// TIA Portal V17 export
// export: Created 2024-09-02T12:50:16.2754473Z, ExportSetting WithDefaults, DisplayName Totally Integrated Automation Portal, DisplayVersion V17, DisplayName TIA Portal Openness, DisplayVersion V17, DisplayName TIA Portal Version Control Interface, DisplayVersion V17, DisplayName STEP 7 Professional, DisplayVersion V17, DisplayName STEP 7 Safety, DisplayVersion V17, DisplayName WinCC Professional, DisplayVersion V17
DATA_BLOCK "AnwDB_ZP_Alarm_OP70"   // DB255
{ S7_Optimized_Access := 'TRUE'; DB_Accessible_From_OPC_UA := 'FALSE' }
AUTHOR : OlegFuehrus
FAMILY : BA
NAME : BA
VERSION : 0.1
// stored: AutoNumber false, DBAccessibleFromOPCUA false, IsOnlyStoredInLoadMemory false, IsRetainMemResEnabled false, IsWriteProtectedInAS false, MemoryReserve 100
   VAR
      FAULT : Array[1..1024] of Bool;
      WARNING : Array[1..1024] of Bool;
      INFORMATION : Array[1..256] of Bool;
      FaultsNo_ST1 : Int;
      FaultsNoSK_ST1 : Int;
      ReportsNo_ST1 : Int;
      FaultsNo_ST2 : Int;
      FaultsNoSK_ST2 : Int;
      ReportsNo_ST2 : Int;
      FaultsNo_ST3 : Int;
      FaultsNoSK_ST3 : Int;
      ReportsNo_ST3 : Int;
   END_VAR
BEGIN
   // FAULT[1] : ESB: Steuerspannung fehlt [+S01- BG0.1]] / Alarm 1: Controle Voltage Not OK [+S01- BG0.1]] / Alarm 1: Stuurspanning niet in(+S01-600KF0.1 of +S01-111KF3) [+S01- BG0.1]]
   // FAULT[2] : ESB: Profibus-Teilnehmer gestört
   // FAULT[3] : ESB: ProfiNet-Teilnehmer gestört / Alarm 3: ProfiNet - Member fault / Alarm 3: ProfiNet - Deelnemerfout
   // FAULT[4] : ESB: Einschaltbedingung fehlt / Alarm 4: switch-on condition missing / Alarm 4: Inschakelvoorwaarde ontbreekt
   // FAULT[5] : ESB: Pneumatikdruck n.i.O. [+M01- BG50.7] / Alarm 5: Pneumatic pressure on OP70 NIO [+M01- BG50.7] / Alarm 5: Pneumatische druk OP70 NIO [+M01- BG50.7]
   // FAULT[6] : ESB: Sicherungsfall 24V [ -100TB1-100FC3/6/8 , [+S01- BG0.2]] / Alarm 6: 24V fuse fault [ -100TB1-100FC3/6/8 , [+S01- BG0.2]] / Alarm 6: 24V-zekeringfout [ -100TB1-100FC3/6/8 , [+S01- BG0.2]]
   // FAULT[7] : ESB: Sicherungsfall 230V [-33FC1/-33FB4/6 -44FC1/3, [+S01- BG0.3]] / Alarm 7: 230V fuse fault [-33FC1/-33FB4/6 -44FC3,-45FC1/3/5, [+S01- BG0.3]] / Alarm 7: 230V-zekeringfout [-33FC1/-33FB4/6 -44FC3,-45FC1/3/5, [+S01- BG0.3]]
   // FAULT[8] : ESB: Sicherungsfall 400V [-30QB7-50QB3,[+S01- BG0.4]] / Alarm 8: 400V fuse fault [-30QB7, [+S01- BG0.4]] / Alarm 8: 400V-zekeringfout[-30QB7, [+S01- BG0.4]]
   // FAULT[9] : ESB: Sicherungsfall 230V ....... [+S-QBxxx]
   // FAULT[10] : ESB: Sicherungsfall 230V ....... [+S-QBxxx]
   // FAULT[11] : ESB: kein Text
   // FAULT[12] : ESB: kein Text
   // FAULT[13] : ESB: kein Text
   // FAULT[14] : ESB: kein Text
   // FAULT[15] : ESB: kein Text
   // FAULT[16] : ESB: kein Text
   // FAULT[17] : ESB: kein Text
   // FAULT[18] : ESB: kein Text
   // FAULT[19] : ESB: kein Text
   // FAULT[20] : ESB: kein Text
   // FAULT[21] : ESB: kein Text
   // FAULT[22] : ESB: kein Text
   // FAULT[23] : ESB: kein Text
   // FAULT[24] : ESB: kein Text
   // FAULT[25] : Allg: Nacharbeit in Station aktiv / Alarm 25: Reworking in Station / Alarm 25: Rework in Station
   // FAULT[26] : Allg: Moby 1 Störung VorStopper [+M01-17BX1] / Alarm 26: RFID 1 fault prestopper [+M01-17BX1] / Alarm 26: Voorstopper RFID 1 fout [+M01-17BX1]
   // FAULT[27] : Allg: Moby 2 Störung Stopper [+M01-17BX2] / Alarm 27: RFID 2 fault Stopper [+M01-17BX2] / Alarm 27: Stopper RFID 2 fout [+M01-17BX2]
   // FAULT[28] : Allg: Moby 3 Störung Stopper [+M01-17BX2] / Alarm 28: RFID 3 fault Stopper [+M01-17BX2] / Alarm 28: Stopper RFID 3 fout [+M01-17BX2]
   // FAULT[29] : Allg: Moby 4 Störung Stopper XXXXX [+M01-BX606]
   // FAULT[30] : Allg: Moby 5 Störung Stopper XXXXX [+M01-BX608]
   // FAULT[31] : Allg: Moby 6 Störung Stopper XXXXX [+M01-BX610]
   // FAULT[32] : Allg: kein Text
   // FAULT[33] : Allg: Pneumatikdruck n.i.O. Station [+M01 - BG700.0/1] / Alarm 33: Central Pneumatic fault [+M01- BG50.7] / Alarm 33: Pneumatische toevoer storing OP70 [+M01- BG50.7]
   // FAULT[34] : Allg: Pneumatikdruck n.i.O. Roboter 1 [+M01 - BG707.0/1] / Alarm 34: Pneumatic ON Gripper fault [+M01- BG53.7] / Alarm 34: Pneumatische toevoer storing OP70 - grijper [+M01- BG53.7]
   // FAULT[35] : Allg: Pneumatikdruck n.i.O. Roboter 2 [+M01 - BG707.2/3]
   // FAULT[36] : Allg: Pneumatikdruck n.i.O. Reserve
   // FAULT[37] : Allg: kein Text
   // FAULT[38] : Allg: kein Text
   // FAULT[39] : Allg: kein Text
   // FAULT[40] : Allg: kein Text
   // FAULT[41] : Allg: kein Text
   // FAULT[42] : Allg: Temperatur Schaltschrank (>30 Minuten) überschritten [+S01--300BT0.7] / Alarm 42: Control cabinet temperature exceeded (> 30 minutes) [+S01--300BT0.7] / Alarm 42: Temperatuur schakelkast overschreden (> 30 minuten) [+S01--300BT0.7]
   // FAULT[43] : Allg: kein Text
   // FAULT[44] : Allg: kein Text
   // FAULT[45] : Allg: Alarm Netzgerät vor Maschine Ein [+S01-600KF0.1] / Alarm 45: Power supply in Machine On Alarm [+S01-600KF0.1] / Alarm 45: Stuurspanning niet in [+S01-600KF0.1]
   // FAULT[46] : Allg: Störung ProfiNet Switch -275XF1 [+S01- BG0.5] / Alarm 46: Fault in ProfiNet Switch -275XF1 [+S01- BG0.5] / Alarm 46: Storing in ProfiNet Switch -275XF1 [+S01- BG0.5]
   // FAULT[47] : Allg: kein Text
   // FAULT[48] : Allg: Grundstellungsfahrt erforderlich / Alarm 48: Home required not allowed / Alarm 48: HOME positie rijden niet toegestaan
   // FAULT[49] : Safety: NOT-HALT Hauptbedienpult OP 40 gestört [+ZP01-302SF30.0] / Alarm 49: EMERGENCY STOP Main Panel OP70[+ZP01-302SF30.0] / Alarm 49: NOODSTOP HMI OP 70[+ZP01-302SF30.0]
   // FAULT[50] : Safety: NOT-HALT Hauptbedienpult OP 50 gestört [+ZP01-11SF5] / Alarm 50: EMERGENCY STOP Main Panel OP 50[+ZP01-11SF5] / Alarm 50: NOODSTOP HMI OP 70[+ZP01-11SF5]
   // FAULT[51] : Safety: NOT-HALT Schutztür XXXXXX gestört [+M01-SF320]
   // FAULT[52] : Safety: NOT-HALT Schutztür XXXXXX gestört [+M01-SF 340]
   // FAULT[53] : Safety: NOT-HALT Roboter 1 gestört [+R01-SF 1]
   // FAULT[54] : Safety: NOT-HALT Roboter 2 gestört [+R02-SF 1]
   // FAULT[55] : Safety: NOT-HALT Reserve
   // FAULT[56] : Safety: NOT-HALT Reserve
   // FAULT[57] : Safety: NOT-HALT Reserve
   // FAULT[58] : Safety: NOT-HALT Reserve
   // FAULT[59] : Safety: NOT-HALT Reserve
   // FAULT[60] : Safety: NOT-HALT Reserve
   // FAULT[61] : Safety: NOT-HALT Reserve
   // FAULT[62] : Safety: NOT-HALT Reserve
   // FAULT[63] : Safety: NOT-HALT Reserve
   // FAULT[64] : Safety: NOT-HALT nicht quittiert OP40 / Alarm 64: EMERGENCY STOP MAIN PANEL OP70 not acknowledged / Alarm 64: NOODSTOP HMI OP 70 niet bevestigd
   // FAULT[65] : Safety: NOT-HALT nicht quittiert OP50 / Alarm 65: EMERGENCY STOP MAIN PANEL OP50 not acknowledged / Alarm 65: NOODSTOP HMI OP70 niet bevestigd
   // FAULT[66] : Safety: Schutztür Station offen [+M01-30SF0] / Alarm 66: Safety Door opened [+M01-260SF2] / Alarm 66: Veiligheidsdeur geopend OP70 [+M01-260SF0]
   // FAULT[67] : Safety: Schutztür Station offen [+M01-SF210.1]
   // FAULT[68] : Safety: Schutztür Station offen [+M01-SFxxxx]
   // FAULT[69] : Safety: Schutztür Reserve
   // FAULT[70] : Safety: Schutztür Reserve
   // FAULT[71] : Safety: Schutztür Reserve
   // FAULT[72] : Safety: Schutztür Reserve
   // FAULT[73] : Safety: Schutztür Reserve
   // FAULT[74] : Safety: Schutztür Reserve
   // FAULT[75] : Safety: Schutztür Reserve
   // FAULT[76] : Safety: Schutztür Reserve
   // FAULT[77] : Safety: Schutztür Reserve
   // FAULT[78] : Safety: Schutztür Reserve
   // FAULT[79] : Safety: Schutztür Reserve
   // FAULT[80] : Safety: Schutztür Reserve
   // FAULT[81] : Safety: Schutztür Station nicht quittiert
   // FAULT[82] : Safety: Schutztür Station nicht quittiert
   // FAULT[83] : Safety: Schutztür Station nicht quittiert / Alarm 83: Safety Door not acknowledged / Alarm 83: Veiligheidsdeur gesloten OP70 niet bevestigd
   // FAULT[84] : Safety: Lichtgitter WT Einlauf ausgelöst (Muting)
   // FAULT[85] : Safety: Lichtgitter WT Auslauf ausgelöst (Muting)
   // FAULT[86] : Safety: Lichtgitter Reserve
   // FAULT[87] : Safety: Lichtgitter Reserve
   // FAULT[88] : Safety: Lichtgitter Reserve
   // FAULT[89] : Safety: Lichtgitter Reserve
   // FAULT[90] : Alarm 90: Safety Bolts Sensor not active, Bolts insite / Alarm 90: Sensor veiligheidsbouten niet actief, bouten op locatie
   // FAULT[91] : Safety: Lichtgitter Reserve
   // FAULT[92] : Safety: Lichtgitter Reserve
   // FAULT[93] : Safety: Lichtgitter Reserve
   // FAULT[94] : Safety: Lichtgitter Reserve
   // FAULT[95] : Safety: Lichtgitter Reserve
   // FAULT[96] : Safety: Lichtgitter Reserve
   // FAULT[97] : Safety: Lichtgitter WT Einlauf nicht quittiert (Muting)
   // FAULT[98] : Safety: Lichtgitter WT Auslauf nicht quittiert (Muting)
   // FAULT[99] : Safety: Freigabekreise gestört
   // FAULT[100] : Safety: Freigabekreis 1 gestört - Medien einschalten
   // FAULT[101] : Safety: Freigabekreis 1 gestört - Sicherheit Station NIO / Alarm 101: Safety Feedback Circuit 1 - Enabling safety Circuit OP70 NOK / Alarm 101: Veiligheidsfeedbackcircuit 1 - inschakelen van veiligheidscircuit OP70 NOK
   // FAULT[102] : Safety: Freigabekreis 2 gestört - Not Halt NIO / Alarm 102: Safety Feedback Circuit 2 - Enabling safety Circuit 2(Emergency stop) NOK / Alarm 102: Veiligheidsfeedbackcircuit 2 - inschakelen van veiligheidscircuit 2 (noodstop) NOK
   // FAULT[103] : Safety: Freigabekreis 4 gestört -
   // FAULT[104] : Safety: Freigabekreis 5 gestört -
   // FAULT[105] : Safety: Freigabekreis 6 gestört -
   // FAULT[106] : Safety: Freigabekreis 7 gestört -
   // FAULT[107] : Safety: Freigabekreis 8 gestört -
   // FAULT[108] : Safety: Freigabekreis 9 gestört -
   // FAULT[109] : Safety: Freigabekreis 10 gestört -
   // FAULT[110] : Safety: Freigabekreis 11 gestört -
   // FAULT[111] : Safety: Freigabekreis 12 gestört -
   // FAULT[112] : Safety: Freigabekreis 13 gestört -
   // FAULT[113] : Safety: Freigabekreis 14 gestört
   // FAULT[114] : Safety: Freigabekreis 15 gestört
   // FAULT[115] : Safety: F-Baugruppenfehler: "F00030_-265KF5".QBAD / Alarm 115: Module error: "F00030_-265KF5".QBAD / Alarm 115: Profisafeodulefout: "F00030_-265KF5".QBAD
   // FAULT[116] : Safety: F-Baugruppenfehler: "F00036_-265KF6".QBAD / Alarm 116: Module error: "F00036_-265KF6".QBAD / Alarm 116: Profisafe modulefout: "F00036_-265KF6".QBAD
   // FAULT[117] : Safety: F-Baugruppenfehler: Reserve
   // FAULT[118] : Safety: F-Baugruppenfehler: Reserve
   // FAULT[119] : Safety: F-Baugruppenfehler: Reserve
   // FAULT[120] : Safety: F-Baugruppenfehler: Reserve
   // FAULT[121] : Safety: F-Baugruppenfehler: Reserve
   // FAULT[122] : Safety: F-Baugruppenfehler: Reserve
   // FAULT[123] : Safety: F-Baugruppenfehler: Reserve
   // FAULT[124] : Safety: F-Baugruppenfehler: Reserve
   // FAULT[125] : Safety: F-Baugruppenfehler: Reserve
   // FAULT[126] : Safety: F-Baugruppenfehler: Reserve
   // FAULT[127] : Safety: F-Baugruppenfehler: Reserve
   // FAULT[128] : Safety: F-Baugruppenfehler: Reserve
   // FAULT[129] : Safety: F-Baugruppenfehler: Reserve
   // FAULT[130] : Safety: F-Baugruppenfehler: Reserve
   // FAULT[131] : Safety: F-Baugruppenfehler: Reserve
   // FAULT[132] : Safety: F-Baugruppenfehler: Reserve
   // FAULT[133] : Safety: F-Baugruppenfehler: Reserve
   // FAULT[134] : Safety: F-Baugruppenfehler: Reserve
   // FAULT[135] : Safety: F-Baugruppenfehler: Reserve
   // FAULT[136] : Safety: F-Baugruppenfehler: Reserve
   // FAULT[137] : Safety: F-Baugruppenfehler: Reserve
   // FAULT[138] : Safety: F-Baugruppenfehler: Reserve
   // FAULT[139] : Safety: F-Baugruppenfehler: Reserve
   // FAULT[140] : Safety: F-Baugruppenfehler: Reserve
   // FAULT[141] : Safety: F-Baugruppenfehler: Reserve
   // FAULT[142] : Safety: F-Baugruppenfehler: Reserve
   // FAULT[143] : Safety: F-Baugruppenfehler: Reserve
   // FAULT[144] : Safety: kein Text
   // FAULT[145] : Safety: kein Text
   // FAULT[146] : Safety: kein Text
   // FAULT[147] : Safety: kein Text
   // FAULT[148] : Safety: kein Text
   // FAULT[149] : Safety: kein Text
   // FAULT[150] : Safety: kein Text
   // FAULT[151] : Safety: kein Text
   // FAULT[152] : Safety: kein Text
   // FAULT[153] : Safety: kein Text
   // FAULT[154] : Safety: kein Text
   // FAULT[155] : Safety: kein Text
   // FAULT[156] : Safety: kein Text
   // FAULT[157] : Safety: kein Text
   // FAULT[158] : Safety: kein Text
   // FAULT[159] : Safety: kein Text
   // FAULT[160] : Safety: Schutztür Reserve
   // FAULT[161] : Safety: kein Text
   // FAULT[162] : Safety: kein Text
   // FAULT[163] : Safety: kein Text
   // FAULT[164] : Safety: kein Text
   // FAULT[165] : Safety: kein Text
   // FAULT[166] : Safety: kein Text
   // FAULT[167] : Safety: kein Text
   // FAULT[168] : Safety: kein Text
   // FAULT[169] : Safety: kein Text
   // FAULT[170] : Safety: kein Text
   // FAULT[171] : Safety: kein Text
   // FAULT[172] : Safety: kein Text
   // FAULT[173] : Safety: kein Text
   // FAULT[174] : Safety: kein Text
   // FAULT[175] : Safety: kein Text
   // FAULT[176] : Safety: kein Text
   // FAULT[177] : Safety: Rückführkreisüberwachung Sicherheit Station NIO [E3.4] / Alarm 177: Feedback circuit monitoring Enabling safety Circuit 1 OP70 [+S01- BG3.4] / Alarm 177: Bewaking terugkoppelingscircuit veiligheid station OK OP70[+S01- BG3.4]
   // FAULT[178] : Safety: Rückführkreisüberwachung Not Halt NIO [E3.5] / Alarm 178: Feedback circuit monitoring EMERGENCY STOP Station [E3.5] / Alarm 178: Bewaking terugkoppelingscircuit noodstop OK OP70 [E3.5]
   // FAULT[179] : Safety: Rückführkreisüberwachung Luft NIO [E50.7] / Alarm 179: Feedback circuit monitoring Pneumatic NOK [+M01- BG50.7] / Alarm 179: Bewaking terugkoppelcircuit Pneumatisch NOK[+M01- BG50.7]
   // FAULT[180] : Safety: Rückführkreisüberwachung Luft im Greifer NIO [E53.7] / Alarm 180: Feedback circuit monitoring Pneumatic NOK in Gripper [+M01- BG53.7] / Alarm 180: Bewaking terugkoppelcircuit Pneumatisch NOK in grijper[+M01- BG53.7]
   // FAULT[181] : Safety: Rückführkreisüberwachung Reserve
   // FAULT[182] : Safety: Rückführkreisüberwachung Reserve
   // FAULT[183] : Safety: Rückführkreisüberwachung Reserve
   // FAULT[184] : Safety: Rückführkreisüberwachung mPro400SG fehlerhaft [E3.2]
   // FAULT[185] : Safety: Rückführkreisüberwachung Reserve
   // FAULT[186] : Safety: Rückführkreisüberwachung Vertikalachse Bremsen [QL712.0/1]
   // FAULT[187] : Safety: Rückführkreisüberwachung Reserve
   // FAULT[188] : Safety: Rückführkreisüberwachung Reserve
   // FAULT[189] : Safety: Rückführkreisüberwachung Reserve
   // FAULT[190] : Alarm 190: Feeder Unit Empty Damper Cap [I55.4] / Alarm 190: Demperdop van de invoereenheid leeg [I55.4]
   // FAULT[191] : Alarm 191: Feeder Unit Empty Ball [I56.0] / Alarm 191: Lege bal invoereenheid [I56.0]
   // FAULT[192] : Alarm 192: Feeder Unit Empty Screw [I56.1] / Alarm 192: Schroef invoereenheid leeg [I56.1]
   // FAULT[193] : Safety: Rückführkreisüberwachung Reserve
   // FAULT[194] : Safety: Rückführkreisüberwachung Reserve
   // FAULT[195] : Safety: Rückführkreisüberwachung Reserve
   // FAULT[196] : Safety: Rückführkreisüberwachung Reserve
   // FAULT[197] : Safety: Rückführkreisüberwachung Reserve
   // FAULT[198] : Safety: Rückführkreisüberwachung Reserve
   // FAULT[199] : Safety: Rückführkreisüberwachung Reserve
   // FAULT[200] : Safety: Rückführkreisüberwachung Reserve
   // FAULT[201] : Safety: Rückführkreisüberwachung Reserve
   // FAULT[202] : Safety: Rückführkreisüberwachung Reserve
   // FAULT[203] : Safety: Rückführkreisüberwachung Reserve
   // FAULT[204] : Safety: Rückführkreisüberwachung Reserve
   // FAULT[205] : Safety: Rückführkreisüberwachung Reserve
   // FAULT[206] : Safety: Rückführkreisüberwachung Reserve
   // FAULT[207] : Safety: Rückführkreisüberwachung Reserve
   // FAULT[208] : Safety: Rückführkreisüberwachung Reserve
   // FAULT[209] : Fehler Schmierzyklus - Automatik gesperrt
   // FAULT[210] : Allg: kein Text
   // FAULT[211] : Allg: kein Text
   // FAULT[212] : Allg: kein Text
   // FAULT[213] : Allg: kein Text
   // FAULT[214] : Allg: kein Text
   // FAULT[215] : Allg: kein Text
   // FAULT[216] : Allg: kein Text
   // FAULT[217] : Allg: kein Text
   // FAULT[218] : Allg: kein Text
   // FAULT[219] : Allg: kein Text
   // FAULT[220] : Allg: kein Text
   // FAULT[221] : Allg: kein Text
   // FAULT[222] : Allg: kein Text
   // FAULT[223] : Allg: kein Text
   // FAULT[224] : Allg: kein Text
   // FAULT[225] : Allg: kein Text
   // FAULT[226] : Allg: kein Text
   // FAULT[227] : Allg: kein Text
   // FAULT[228] : Allg: kein Text
   // FAULT[229] : Allg: kein Text
   // FAULT[230] : Allg: kein Text
   // FAULT[231] : Allg: kein Text
   // FAULT[232] : Allg: kein Text
   // FAULT[233] : Allg: kein Text
   // FAULT[234] : Allg: kein Text
   // FAULT[235] : Allg: kein Text
   // FAULT[236] : Allg: kein Text
   // FAULT[237] : Allg: kein Text
   // FAULT[238] : Allg: kein Text
   // FAULT[239] : Allg: kein Text
   // FAULT[240] : Allg: kein Text
   // FAULT[241] : Allg: kein Text
   // FAULT[242] : Allg: kein Text
   // FAULT[243] : Allg: kein Text
   // FAULT[244] : Allg: kein Text
   // FAULT[245] : Allg: kein Text
   // FAULT[246] : Allg: kein Text
   // FAULT[247] : Allg: kein Text
   // FAULT[248] : Allg: kein Text
   // FAULT[249] : Allg: kein Text
   // FAULT[250] : Allg: kein Text
   // FAULT[251] : Allg: kein Text
   // FAULT[252] : Allg: kein Text
   // FAULT[253] : Allg: kein Text
   // FAULT[254] : Allg: kein Text
   // FAULT[255] : Allg: kein Text
   // FAULT[256] : Allg: kein Text
   // FAULT[257] : Allg: kein Text
   // FAULT[258] : Allg: kein Text
   // FAULT[259] : Allg: kein Text
   // FAULT[260] : Allg: kein Text
   // FAULT[261] : Allg: kein Text
   // FAULT[262] : Allg: kein Text
   // FAULT[263] : Allg: kein Text
   // FAULT[264] : Allg: kein Text
   // FAULT[265] : Überwachung Schütz "Sinamics" nicht abgefallen bzw. defeckt (+S01-QA101.1)
   // FAULT[266] : Überwachung Schütz "Kühlgerät" nicht abgefallen bzw. defeckt (+S01-QA100.2)
   // FAULT[267] : Überwachung Schütz "Schmierung" nicht abgefallen bzw. defeckt (+S01-QA101.0)
   // FAULT[268] : Überwachung Schütz "Schraubtechnik" nicht abgefallen bzw. defeckt (+S01-QA102.0)
   // FAULT[269] : Überwachung Schütz " " nicht abgefallen Reserve
   // FAULT[270] : Überwachung Schütz " " nicht abgefallen Reserve
   // FAULT[271] : Überwachung Schütz " " nicht abgefallen Reserve
   // FAULT[272] : Überwachung Schütz " " nicht abgefallen Reserve
   // FAULT[273] : Überwachung Schütz " " nicht abgefallen Reserve
   // FAULT[274] : Überwachung Schütz " " nicht abgefallen Reserve
   // FAULT[275] : Allg: kein Text
   // FAULT[276] : Allg: kein Text
   // FAULT[277] : Allg: kein Text
   // FAULT[278] : Allg: kein Text
   // FAULT[279] : Allg: kein Text
   // FAULT[280] : Allg: kein Text
   // FAULT[281] : Allg: kein Text
   // FAULT[282] : Allg: kein Text
   // FAULT[283] : Allg: kein Text
   // FAULT[284] : Allg: kein Text
   // FAULT[285] : Allg: kein Text
   // FAULT[286] : Allg: kein Text
   // FAULT[287] : Allg: kein Text
   // FAULT[288] : Allg: kein Text
   // FAULT[289] : Allg: kein Text
   // FAULT[290] : Allg: kein Text
   // FAULT[291] : Allg: kein Text
   // FAULT[292] : Allg: kein Text
   // FAULT[293] : Allg: kein Text
   // FAULT[294] : Allg: kein Text
   // FAULT[295] : Allg: kein Text
   // FAULT[296] : Allg: kein Text
   // FAULT[297] : Serienfehler: BEA1 Lagerrahmen verschrauben - Schraubstelle 01 / SeriesError: FG01 BEA1 Assembly Damper Cap / Seriefout: FG01 BEA1 Montage demper cap
   // FAULT[298] : Serienfehler: BEA1 Lagerrahmen verschrauben - Schraubstelle 02 / SeriesError: FG01 BEA1 Assembly Ball / Seriefout: FG01 BEA1 Montage bal
   // FAULT[299] : Serienfehler: BEA1 Lagerrahmen verschrauben - Schraubstelle 03 / SeriesError: FG01 BEA2 Damper Cap controle / Seriefout: FG01 BEA2 Controle positie demper cap
   // FAULT[300] : Serienfehler: BEA1 Lagerrahmen verschrauben - Schraubstelle 04 / SeriesError: FG02 BEA1 Controle Damper 1 - OP50 / Seriefout: FG02 BEA1 Controle Demper 1 - OP50
   // FAULT[301] : Serienfehler: BEA1 Lagerrahmen verschrauben - Schraubstelle 05 / SeriesError: FG02 BEA1 Controle Damper 2 - OP50 / Seriefout: FG02 BEA1 Controle Demper 2 - OP50
   // FAULT[302] : Serienfehler: BEA1 Lagerrahmen verschrauben - Schraubstelle 06 / SeriesError: FG02 BEA1 Controle Damper 3 - OP50 / Seriefout: FG02 BEA1 Controle Demper 3 - OP50
   // FAULT[303] : Serienfehler: BEA1 Lagerrahmen verschrauben - Schraubstelle 07 / SeriesError: FG02 BEA1 Controle Filter - OP60 / Seriefout: FG02 BEA1 Controle filter - OP60
   // FAULT[304] : Serienfehler: BEA1 Lagerrahmen verschrauben - Schraubstelle 08 / SeriesError: FG02 BEA1 Controle Ball - OP70_1 / Seriefout: FG02 BEA1 Controle kogel - OP70_1
   // FAULT[305] : Serienfehler: BEA1 Lagerrahmen verschrauben - Schraubstelle 09 / SeriesError: FG02 BEA1 Controle Damper Cap - OP70_1 / Seriefout: FG02 BEA1 Controle Demper cap - OP70_1
   // FAULT[306] : Serienfehler: BEA1 Lagerrahmen verschrauben - Schraubstelle 10 / SeriesError: FG02 BEA1 ControleDowel 1 - OP60 / Seriefout: FG02 BEA2 Tussenplaat nemen
   // FAULT[307] : Serienfehler: BEA1 Lagerrahmen verschrauben - Schraubstelle 11 / SeriesError: FG02 BEA1 Controle Dowel 2 - OP60 / Seriefout: FG02 BEA2 Tussenplaat plaatsen
   // FAULT[308] : Serienfehler: BEA1 Lagerrahmen verschrauben - Schraubstelle 12 / SeriesError: FG02 BEA2 Pick Intermediate plate / Seriefout: FG02 BEA3 Tussenplaat vastdraaien
   // FAULT[309] : Serienfehler: BEA1 Lagerrahmen verschrauben - Schraubstelle 13 / SeriesError: FG02 BEA2 Place Intermediate plate
   // FAULT[310] : Serienfehler: BEA1 Lagerrahmen verschrauben - Schraubstelle 14 / SeriesError: FG02 BEA3 Tightening Intermediate plate
   // FAULT[311] : Serienfehler: BEA1 Lagerrahmen verschrauben - Schraubstelle 15
   // FAULT[312] : Serienfehler: BEA1 Lagerrahmen verschrauben - Schraubstelle 16
   // FAULT[313] : Serienfehler: BEA1 Lagerrahmen verschrauben - Schraubstelle 01
   // FAULT[314] : Serienfehler: BEA1 Lagerrahmen verschrauben - Schraubstelle 01
   // FAULT[315] : Serienfehler: Reserve
   // FAULT[316] : Serienfehler: Reserve
   // FAULT[317] : Serienfehler: Reserve
   // FAULT[318] : Serienfehler: Reserve
   // FAULT[319] : Serienfehler: Reserve
   // FAULT[320] : Serienfehler: Reserve
   // FAULT[321] : Serienfehler: Reserve
   // FAULT[322] : Serienfehler: Reserve
   // FAULT[323] : Serienfehler: Reserve
   // FAULT[324] : Serienfehler: Reserve
   // FAULT[325] : Serienfehler: Reserve
   // FAULT[326] : Serienfehler: Reserve
   // FAULT[327] : Serienfehler: Reserve
   // FAULT[328] : Serienfehler: Reserve
   // FAULT[329] : Allg: kein Text
   // FAULT[330] : Allg: kein Text
   // FAULT[331] : Allg: kein Text
   // FAULT[332] : Allg: kein Text
   // FAULT[333] : Allg: kein Text
   // FAULT[334] : Allg: kein Text
   // FAULT[335] : Allg: kein Text
   // FAULT[336] : Allg: kein Text
   // FAULT[337] : Allg: kein Text
   // FAULT[338] : Allg: kein Text
   // FAULT[339] : Allg: kein Text
   // FAULT[340] : Allg: kein Text
   // FAULT[341] : Paarfehler: MM30/31 Hub-index unten/oben(+M01-BG51.1/51.0) / Pair error: MM30/31 Index Up / Down(+M01-BG51.1/51.0) / Paarfout: MM30/31 Index Boven/Onder (+M01-BG51.1/51.0)
   // FAULT[342] : Paarfehler: MM50/51 Hub-index unten/oben(+M01-BG51.3-5/51.2-4) / Pair error: MM50/51 Index Up / Down(+M01-BG51.3-5/51.2-4) / Paarfout: MM50/51 Index Boven/Onder (+M01-BG51.3-5/51.2-4)
   // FAULT[343] : Paarfehler: MM70/71 Hub-index unten/oben(+M01-BG52.0/52.1) / Pair error: MM70/71 Index Up / Down(+M01-BG52.0/52.1) / Paarfout: MM70/71 Index Boven/Onder (+M01-BG52.0/52.1)
   // FAULT[344] : Pair error: MM110 Sliding Damper Cap Back/ Front (+M01-BG52.5/4) / Paarfehler: MM110 Schieber Kappe züruck/vor (+M01-BG52.5/4) / Paarfout: MM110 schuifdemperkap Vooraan/Achteraan (+M01-BG52.5/4)
   // FAULT[345] : Paarfehler: MM120 Schieber Kugel züruck/vor (+M01-BG53.0/1) / Pair error: MM120 Sliding Ball Back/ Front (+M01-BG53.0/1) / Paarfout: MM120 Sliding Ball Vooraan/Achteraan (+M01-BG53.0/1)
   // FAULT[346] : Paarfehler: MM130 Fügeeinheit Kappe senken/heben(+M01-BG53.3/4) / Pair error: MM130 Press Damper Cap Up/Down (+M01-BG53.3/4) / Paarfout: MM130 Druk demperkap Boven/Onder (+M01-BG53.3/4)
   // FAULT[347] : Paarfehler: MM140 Y-Achse Übersetzer züruck/vor(+M01-BG53.5/6) / Pair error: MM140 Y-Axis Gripper Back/ Front (+M01-BG53.5/6) / Paarfout: MM140 Y-as grijper Vooraan/Achteraan(+M01-BG53.5/6)
   // FAULT[348] : Paarfehler: MM160 Z-Achse Übersetzerl heben/senken (+M01-BG54.0/1) / Pair error: MM150 Z-Axis Gripper Up/Down (+M01-BG54.0/1) / Paarfout: MM150 Z-as grijper Boven/Onder (+M01-BG54.0/1)
   // FAULT[349] : Paarfehler: MM170 Hubzylinder Schraubeinheit heben/senken(+M01-BG54.2/3) / Pair error: MM160 Z-Axis Screwdriver Up/Down (+M01-BG54.2/3) / Paarfout: MM160 Z-as schroevendraaier Boven/Onder (+M01-BG54.2/3)
   // FAULT[350] : Paarfehler: MM180 Zustellschlitten heben/senken (+M01-BG54.4/5) / Pair error: MM170 Z-Axis Screwdriver unit Up/Down (+M01-BG54.4/5) / Paarfout: MM170 Z-as Schroevendraaiereenheid Boven/Onder (+M01-BG54.4/5)
   // FAULT[351] : Paarfehler: MM200 Übersetzen Hülse züruck/vor (+M01-BG63.0/1) / Pair error: MM210 Loading cylinder Dumper Cap Up/Down (+M01-BG55.0/1) / Paarfout: MM210 Laadcilinder Dumper Cap Boven/Onder (+M01-BG55.0/1)
   // FAULT[352] : Paarfehler: MM210 Zustellung Hülse züruck/vor (+M01-BG63.2/3) / Pair error: MM220 Separation cylinder Dumper Cap unit front/back (+M01-BG55.6/7) / Paarfout: MM220 Scheidingscilinder Dumper Cap unit Vooraan/Achteraan (+M01-BG55.6/7)
   // FAULT[353] : Paarfehler: *** reserviert für Paarfehler ***
   // FAULT[354] : Paarfehler: *** reserviert für Paarfehler ***
   // FAULT[355] : Paarfehler: *** reserviert für Paarfehler ***
   // FAULT[356] : Paarfehler: *** reserviert für Paarfehler ***
   // FAULT[357] : Paarfehler: *** reserviert für Paarfehler ***
   // FAULT[358] : Paarfehler: *** reserviert für Paarfehler ***
   // FAULT[359] : Paarfehler: *** reserviert für Paarfehler ***
   // FAULT[360] : Paarfehler: *** reserviert für Paarfehler ***
   // FAULT[361] : Paarfehler: *** reserviert für Paarfehler ***
   // FAULT[362] : Paarfehler: *** reserviert für Paarfehler ***
   // FAULT[363] : Paarfehler: *** reserviert für Paarfehler ***
   // FAULT[364] : Paarfehler: *** reserviert für Paarfehler ***
   // FAULT[365] : Paarfehler: *** reserviert für Paarfehler ***
   // FAULT[366] : Paarfehler: *** reserviert für Paarfehler ***
   // FAULT[367] : Paarfehler: *** reserviert für Paarfehler ***
   // FAULT[368] : Paarfehler: *** reserviert für Paarfehler ***
   // FAULT[369] : Paarfehler: *** reserviert für Paarfehler ***
   // FAULT[370] : Paarfehler: *** reserviert für Paarfehler ***
   // FAULT[371] : Paarfehler: *** reserviert für Paarfehler ***
   // FAULT[372] : Paarfehler: *** reserviert für Paarfehler ***
   // FAULT[373] : Paarfehler: *** reserviert für Paarfehler ***
   // FAULT[374] : Paarfehler: *** reserviert für Paarfehler ***
   // FAULT[375] : Paarfehler: *** reserviert für Paarfehler ***
   // FAULT[376] : Paarfehler: *** reserviert für Paarfehler ***
   // FAULT[377] : Paarfehler: *** reserviert für Paarfehler ***
   // FAULT[378] : Paarfehler: *** reserviert für Paarfehler ***
   // FAULT[379] : Paarfehler: *** reserviert für Paarfehler ***
   // FAULT[380] : Paarfehler: *** reserviert für Paarfehler ***
   // FAULT[381] : Paarfehler: *** reserviert für Paarfehler ***
   // FAULT[382] : Paarfehler: *** reserviert für Paarfehler ***
   // FAULT[383] : Paarfehler: *** reserviert für Paarfehler ***
   // FAULT[384] : Paarfehler: *** reserviert für Paarfehler ***
   // FAULT[385] : Paarfehler: *** reserviert für Paarfehler ***
   // FAULT[386] : Paarfehler: *** reserviert für Paarfehler ***
   // FAULT[387] : Paarfehler: *** reserviert für Paarfehler ***
   // FAULT[388] : Paarfehler: *** reserviert für Paarfehler ***
   // FAULT[389] : Paarfehler: *** reserviert für Paarfehler ***
   // FAULT[390] : Paarfehler: *** reserviert für Paarfehler ***
   // FAULT[391] : Paarfehler: *** reserviert für Paarfehler ***
   // FAULT[392] : Paarfehler: *** reserviert für Paarfehler ***
   // FAULT[393] : Paarfehler: *** reserviert für Paarfehler ***
   // FAULT[394] : Paarfehler: *** reserviert für Paarfehler ***
   // FAULT[395] : Paarfehler: *** reserviert für Paarfehler ***
   // FAULT[396] : Paarfehler: *** reserviert für Paarfehler ***
   // FAULT[397] : Paarfehler: *** reserviert für Paarfehler ***
   // FAULT[398] : Paarfehler: *** reserviert für Paarfehler ***
   // FAULT[399] : Paarfehler: *** reserviert für Paarfehler ***
   // FAULT[400] : Paarfehler: *** reserviert für Paarfehler ***
   // FAULT[401] : Paarfehler: *** reserviert für Paarfehler ***
   // FAULT[402] : Paarfehler: *** reserviert für Paarfehler ***
   // FAULT[403] : Paarfehler: *** reserviert für Paarfehler ***
   // FAULT[404] : Paarfehler: *** reserviert für Paarfehler ***
   // FAULT[405] : Paarfehler: *** reserviert für Paarfehler ***
   // FAULT[406] : Paarfehler: *** reserviert für Paarfehler ***
   // FAULT[407] : Paarfehler: *** reserviert für Paarfehler ***
   // FAULT[408] : Paarfehler: *** reserviert für Paarfehler ***
   // FAULT[409] : Paarfehler: *** reserviert für Paarfehler ***
   // FAULT[410] : Paarfehler: *** reserviert für Paarfehler ***
   // FAULT[411] : Paarfehler: *** reserviert für Paarfehler ***
   // FAULT[412] : Paarfehler: *** reserviert für Paarfehler ***
   // FAULT[413] : Paarfehler: *** reserviert für Paarfehler ***
   // FAULT[414] : Paarfehler: *** reserviert für Paarfehler ***
   // FAULT[415] : Paarfehler: *** reserviert für Paarfehler ***
   // FAULT[416] : Paarfehler: *** reserviert für Paarfehler ***
   // FAULT[417] : Fehler - Automatik gesperrt
   // FAULT[418] : Fehler - Automatik gesperrt
   // FAULT[419] : Fehler - Automatik gesperrt
   // FAULT[420] : Fehler - Automatik gesperrt
   // FAULT[421] : Fehler - Automatik gesperrt
   // FAULT[422] : Fehler - Automatik gesperrt
   // FAULT[423] : Fehler - Automatik gesperrt
   // FAULT[424] : Fehler - Automatik gesperrt
   // FAULT[425] : Achse: Vertikalschlitten - Motorschutz [+S01-QA1.1]
   // FAULT[426] : Achse: Vertikalschlitten - Störung [+S01-KF110]
   // FAULT[427] : Achse: Vertikalschlitten - Bremsentest n.i.O.
   // FAULT[428] : Achse: kein Text
   // FAULT[429] : Achse: kein Text
   // FAULT[430] : Achse: kein Text
   // FAULT[431] : Achse: kein Text
   // FAULT[432] : Achse: kein Text
   // FAULT[433] : Achse: kein Text
   // FAULT[434] : Achse: kein Text
   // FAULT[435] : Achse: kein Text
   // FAULT[436] : Achse: kein Text
   // FAULT[437] : Achse: kein Text
   // FAULT[438] : Achse: kein Text
   // FAULT[439] : Achse: kein Text
   // FAULT[440] : Achse: kein Text
   // FAULT[441] : Achse: kein Text
   // FAULT[442] : Achse: kein Text
   // FAULT[443] : Achse: kein Text
   // FAULT[444] : Achse: kein Text
   // FAULT[445] : Achse: kein Text
   // FAULT[446] : Achse: kein Text
   // FAULT[447] : Achse: kein Text
   // FAULT[448] : Achse: kein Text
   // FAULT[449] : Achse: kein Text
   // FAULT[450] : Achse: kein Text
   // FAULT[451] : Achse: kein Text
   // FAULT[452] : Achse: kein Text
   // FAULT[453] : Achse: kein Text
   // FAULT[454] : Achse: kein Text
   // FAULT[455] : Achse: kein Text
   // FAULT[456] : Achse: kein Text
   // FAULT[457] : Schrauber: MPRO 1 nicht Betriebsbereit [+M-KF100]
   // FAULT[458] : Schrauber: MPRO 1 Sicherungen ausgelöst [E1.4]
   // FAULT[459] : Schrauber: kein Text
   // FAULT[460] : Schrauber: kein Text
   // FAULT[461] : Schrauber: kein Text
   // FAULT[462] : Schrauber: kein Text
   // FAULT[463] : Schrauber: kein Text
   // FAULT[464] : Schrauber: kein Text
   // FAULT[465] : Schrauber: kein Text
   // FAULT[466] : Schrauber: kein Text
   // FAULT[467] : Schrauber: kein Text
   // FAULT[468] : Schrauber: kein Text
   // FAULT[469] : Schrauber: kein Text
   // FAULT[470] : Schrauber: kein Text
   // FAULT[471] : Schrauber: kein Text
   // FAULT[472] : Schrauber: kein Text
   // FAULT[473] : Allg: kein Text
   // FAULT[474] : Allg: kein Text
   // FAULT[475] : Allg: kein Text
   // FAULT[476] : Allg: kein Text
   // FAULT[477] : Allg: kein Text
   // FAULT[478] : Allg: kein Text
   // FAULT[479] : Allg: kein Text
   // FAULT[480] : Allg: kein Text
   // FAULT[481] : Allg: kein Text
   // FAULT[482] : Allg: kein Text
   // FAULT[483] : Allg: kein Text
   // FAULT[484] : Allg: kein Text
   // FAULT[485] : Allg: kein Text
   // FAULT[486] : Allg: kein Text
   // FAULT[487] : Allg: kein Text
   // FAULT[488] : Allg: kein Text
   // FAULT[489] : Allg: kein Text
   // FAULT[490] : Allg: kein Text
   // FAULT[491] : Allg: kein Text
   // FAULT[492] : Allg: kein Text
   // FAULT[493] : Allg: kein Text
   // FAULT[494] : Allg: kein Text
   // FAULT[495] : Allg: kein Text
   // FAULT[496] : Allg: kein Text
   // FAULT[497] : Allg: kein Text
   // FAULT[498] : Allg: kein Text
   // FAULT[499] : Allg: kein Text
   // FAULT[500] : Allg: kein Text / Alarm 500: X2 - The assumed level of NOK has been reached / Alarm 500: X2 - Het ingestelde niveau aantal NOK delen is bereikt
   // FAULT[501] : Allg: kein Text
   // FAULT[502] : Allg: kein Text
   // FAULT[503] : Allg: kein Text
   // FAULT[504] : Allg: kein Text
   // FAULT[505] : Allg: kein Text
   // FAULT[506] : Allg: kein Text
   // FAULT[507] : Allg: kein Text
   // FAULT[508] : Allg: kein Text
   // FAULT[509] : Allg: kein Text
   // FAULT[510] : Allg: kein Text
   // FAULT[511] : Allg: kein Text
   // FAULT[512] : Allg: kein Text
   // FAULT[513] : Roboter 1 - Greiferbewegung verklemmt [+R01]
   // FAULT[514] : Roboter 1 - Kollisionsschutz ausgelöst [+R01]
   // FAULT[515] : Roboter 1 - Fehler Teilekontrolle Greifer 1
   // FAULT[516] : Roboter 1 - Fehler Teilekontrolle Greifer 2
   // FAULT[517] : Roboter 1 -
   // FAULT[518] : Roboter 1 -
   // FAULT[519] : Roboter 1 -
   // FAULT[520] : Roboter 1 -
   // FAULT[521] : Roboter 1 -
   // FAULT[522] : Roboter 1 -
   // FAULT[523] : Roboter 1 -
   // FAULT[524] : Roboter 1 -
   // FAULT[525] : Roboter 1 -
   // FAULT[526] : Roboter 1 -
   // FAULT[527] : Roboter 1 -
   // FAULT[528] : Roboter 1 -
   // FAULT[529] : Roboter 2 - Greiferbewegung verklemmt [+R02]
   // FAULT[530] : Roboter 2 - Kollisionsschutz ausgelöst [+R02]
   // FAULT[531] : Roboter 2 - Fehler Teilekontrolle Greifer 1
   // FAULT[532] : Roboter 2 - Fehler Teilekontrolle Greifer 2
   // FAULT[533] : Roboter 2 -
   // FAULT[534] : Roboter 2 -
   // FAULT[535] : Roboter 2 -
   // FAULT[536] : Roboter 2 -
   // FAULT[537] : Roboter 2 -
   // FAULT[538] : Roboter 2 -
   // FAULT[539] : Roboter 2 -
   // FAULT[540] : Roboter 2 -
   // FAULT[541] : Roboter 2 -
   // FAULT[542] : Roboter 2 -
   // FAULT[543] : Roboter 2 -
   // FAULT[544] : Roboter 2 -
   // FAULT[545] : fehler545
   // FAULT[546] : fehler546
   // FAULT[547] : fehler547
   // FAULT[548] : fehler548
   // FAULT[549] : fehler549
   // FAULT[550] : fehler550
   // FAULT[551] : fehler551
   // FAULT[552] : fehler552
   // FAULT[553] : fehler553
   // FAULT[554] : fehler554
   // FAULT[555] : fehler555
   // FAULT[556] : fehler556
   // FAULT[557] : fehler557
   // FAULT[558] : fehler558
   // FAULT[559] : fehler559
   // FAULT[560] : fehler560
   // FAULT[561] : fehler561
   // FAULT[562] : fehler562
   // FAULT[563] : fehler563
   // FAULT[564] : fehler564
   // FAULT[565] : fehler565
   // FAULT[566] : fehler566
   // FAULT[567] : fehler567
   // FAULT[568] : fehler568
   // FAULT[569] : fehler569
   // FAULT[570] : fehler570
   // FAULT[571] : fehler571
   // FAULT[572] : fehler572
   // FAULT[573] : fehler573
   // FAULT[574] : fehler574
   // FAULT[575] : fehler575
   // FAULT[576] : fehler576
   // FAULT[577] : Kistler -KF121 Fehler im Setup
   // FAULT[578] : Kistler -KF121 Ungültige Werte für die Sensor X-Kalibrierung
   // FAULT[579] : Kistler -KF121 Ungültige Werte für die Sensor Y-Kalibrierung
   // FAULT[580] : Kistler -KF121 Sensortest war Fehlerhaft
   // FAULT[581] : Kistler -KF121 Eingabe für Kraftbereich Piezo zu klein/gross
   // FAULT[582] : Kistler -KF121 Für Messprogramm wurde kein EO parametriert
   // FAULT[583] : Kistler -KF121 Ein deaktiviertes MP wurde angewählt
   // FAULT[584] : Kistler -KF121 NOK in Folge haben die erlaubte Anzahl überschritten
   // FAULT[585] : Kistler -KF121 Anzahl verpasster Messungen überschritten
   // FAULT[586] : Kistler -KF121 Anzahl der NOK Messungen überschritten
   // FAULT[587] : Kistler -KF121 Hüllkurve Trendüberwachung die Trendgrenze erreicht
   // FAULT[588] : Kistler -KF121 DMS-Sensor nicht angeschlossen oder defekt ist
   // FAULT[589] : Kistler -KF121 Digitalausgang wurde kurz geschlossen
   // FAULT[590] : Kistler -KF121 Sensorversorgung 5 V wird nicht eingehalten
   // FAULT[591] : Kistler -KF121 Speisespannung 24 V wird nicht eingehalten
   // FAULT[592] : Kistler -KF121 Zielverzeichnis hat keinen Speicherplatz
   // FAULT[593] : Kistler -KF121 Zwischenpuffer für unterbrochene Verbindungen voll
   // FAULT[594] : Kistler -KF121 Zugriff auf Variable welche nicht benamt wurde
   // FAULT[595] : Kistler -KF121 Servoverstärker kann keine Leistung hinzugeschaltet werden
   // FAULT[596] : Kistler -KF121 mehrere Fahrbefehle zeitgleich ans Messgerät gesendet
   // FAULT[597] : Kistler -KF121 Sequenz-Element Calculator zwischen MessenStart/Stop plaziert
   // FAULT[598] : Kistler -KF121 Sequenz-Element Calculator sollte durch 0 dividieren
   // FAULT[599] : Kistler -KF121 Bewegung mit Weiterschaltung auf Kraft nicht erfolgt, Kraftwert nicht erreicht
   // FAULT[600] : Kistler -KF121 Position liegt ausserhalb der Fahrbereichsgrenze / Alarm 600: iSynchro on Setting = 4 OP70.1 / Alarm 600: iSynchro aan Setting = 4 OP70.1
   // FAULT[601] : Kistler -KF121 Verbindung zum Servoverstärker unterbrochen / Alarm 601: iSynchro on Result = 4 OP70.1 / Alarm 601: iSynchro aan Result = 4 OP70.1
   // FAULT[602] : Kistler -KF121 Servoverstärker hat Fehler detektiert / Alarm 602: iSynchro on Setting = 4 OP70.2 / Alarm 602: iSynchro aan Setting = 4 OP70.2
   // FAULT[603] : Kistler -KF121 Kraftüberwachung für Fahrbewegung wurde überschritten / Alarm 603: iSynchro on Result = 4 OP70.2 / Alarm 603: iSynchro aan Result = 4 OP70.2
   // FAULT[604] : Kistler -KF121 Tippbewegung wurde ausserhalb vom Tippbereich angesteuert / Alarm 604: iSynchro on Setting = 4 OP70.3 / Alarm 604: iSynchro aan Setting = 4 OP70.3
   // FAULT[605] : Kistler -KF121 Bewegung mit Stopp auf externes Signal hat kein Stoppsignal erhalten / Alarm 605: iSynchro on Result = 4 OP70.3 / Alarm 605: iSynchro aan Result = 4 OP70.3
   // FAULT[606] : Kistler -KF121 Fahrbewegung hat Geschwindigkeit 0 mm/s enthalten / Alarm 606: No communication with the MES system / Alarm 606: Geen communicatie met het MES systeem
   // FAULT[607] : Kistler -KF121 Umrechnungsfaktor für analogen Ausgang kann nicht gesetzt werden / Alarm 607: Defaulty Code on Result == 1 - Product ID not registered in database OP70.1 / Alarm 607: Defaulty Code op resultaat == 1 - Product-ID niet geregistreerd in database OP70.1
   // FAULT[608] : Kistler -KF121 Geschwindigkeit Fahrbewegung ausserhalb Grenzen / Alarm 608: Defaulty Code on Result == 2 - Error during MES processing OP70.1 / Alarm 608: Defaulty Code op resultaat == 2 - Fout tijdens MES-verwerking OP70.1
   // FAULT[609] : Kistler -KF121 Geschwindigkeit Tippbewegung ausserhalb Grenzen / Alarm 609: Defaulty Code on Result == 1 - Product ID not registered in database OP70.2 / Alarm 609: Defaulty Code op resultaat == 1 - Product-ID niet geregistreerd in database OP70.2
   // FAULT[610] : Kistler -KF121 Bremsentest fehlerhaft / Alarm 610: Defaulty Code on Result == 2 - Error during MES processing OP70.2 / Alarm 610: Defaulty Code op resultaat == 2 - Fout tijdens MES-verwerking OP70.2
   // FAULT[611] : Kistler -KF121 Unerwarteter Fehler in der Sequenz / Alarm 611: Defaulty Code on Result == 1 - Product ID not registered in database OP70.3 / Alarm 611: Defaulty Code op resultaat == 1 - Product-ID niet geregistreerd in database OP70.3
   // FAULT[612] : Kistler -KF121 Digitaleingang Timeout / Alarm 612: Defaulty Code on Result == 2 - Error during MES processing OP70.3 / Alarm 612: Defaulty Code op resultaat == 2 - Fout tijdens MES-verwerking OP70.3
   // FAULT[613] : Kistler -KF121 Sollwertdaten SPS -> maXYmos senden / Alarm 613: Defaulty Code on Setting == 1 - Product ID not registered in database OP70.1 / Alarm 613: Defaulty Code bij Setting == 1 - Product-ID niet geregistreerd in database OP70.1
   // FAULT[614] : Kistler -KF121 Power On fehlt / Alarm 614: Defaulty Code on Setting == 2 - Error during MES processing OP70.1 / Alarm 614: Defaulty Code bij Setting == 2 - Fout tijdens MES-verwerking OP70.1
   // FAULT[615] : Kistler -KF121 Servoantrieb Betriebsbereit fehlt / Alarm 615: Defaulty Code on Setting == 1 - Product ID not registered in database OP70.2 / Alarm 615: Defaulty Code bij Setting == 1 - Product-ID niet geregistreerd in database OP70.2
   // FAULT[616] : Kistler -KF121 Unzulässiges Programm vorgewählt / Alarm 616: Defaulty Code on Setting == 2 - Error during MES processing OP70.2 / Alarm 616: Defaulty Code bij Setting == 2 - Fout tijdens MES-verwerking OP70.2
   // FAULT[617] : Kistler -KF121 Sicherheitsstatus SMES aktiv / Alarm 617: Defaulty Code on Setting == 1 - Product ID not registered in databaseOP70.3 / Alarm 617: Defaulty Code bij Setting == 1 - Product-ID niet geregistreerd in databaseOP70.3
   // FAULT[618] : Kistler -KF121 Sicherheitsstatus SMST2 aktiv / Alarm 618: Defaulty Code on Setting == 2 - Error during MES processing OP70.3 / Alarm 618: Defaulty Code bij Setting == 2 - Fout tijdens MES-verwerking OP70.3
   // FAULT[619] : Kistler -KF121 Profinet
   // FAULT[620] : Kistler -KF121 Fehler Servocontroller
   // FAULT[621] : Kistler -KF121 Fehler maXYmos
   // FAULT[622] : Kistler -KF121 Leistung nicht aktiv
   // FAULT[623] : Kistler -KF121 Schutzschalter
   // FAULT[624] : Kistler -KF121 Bremsentest
   // FAULT[625] : Kistler -KF122 Fehler im Setup
   // FAULT[626] : Kistler -KF122 Ungültige Werte für die Sensor X-Kalibrierung
   // FAULT[627] : Kistler -KF122 Ungültige Werte für die Sensor Y-Kalibrierung
   // FAULT[628] : Kistler -KF122 Sensortest war Fehlerhaft
   // FAULT[629] : Kistler -KF122 Eingabe für Kraftbereich Piezo zu klein/gross
   // FAULT[630] : Kistler -KF122 Für Messprogramm wurde kein EO parametriert
   // FAULT[631] : Kistler -KF122 Ein deaktiviertes MP wurde angewählt
   // FAULT[632] : Kistler -KF122 NOK in Folge haben die erlaubte Anzahl überschritten
   // FAULT[633] : Kistler -KF122 Anzahl verpasster Messungen überschritten
   // FAULT[634] : Kistler -KF122 Anzahl der NOK Messungen überschritten
   // FAULT[635] : Kistler -KF122 Hüllkurve Trendüberwachung die Trendgrenze erreicht
   // FAULT[636] : Kistler -KF122 DMS-Sensor nicht angeschlossen oder defekt ist
   // FAULT[637] : Kistler -KF122 Digitalausgang wurde kurz geschlossen
   // FAULT[638] : Kistler -KF122 Sensorversorgung 5 V wird nicht eingehalten
   // FAULT[639] : Kistler -KF122 Speisespannung 24 V wird nicht eingehalten
   // FAULT[640] : Kistler -KF122 Zielverzeichnis hat keinen Speicherplatz
   // FAULT[641] : Kistler -KF122 Zwischenpuffer für unterbrochene Verbindungen voll
   // FAULT[642] : Kistler -KF122 Zugriff auf Variable welche nicht benamt wurde
   // FAULT[643] : Kistler -KF122 Servoverstärker kann keine Leistung hinzugeschaltet werden
   // FAULT[644] : Kistler -KF122 mehrere Fahrbefehle zeitgleich ans Messgerät gesendet
   // FAULT[645] : Kistler -KF122 Sequenz-Element Calculator zwischen MessenStart/Stop plaziert
   // FAULT[646] : Kistler -KF122 Sequenz-Element Calculator sollte durch 0 dividieren
   // FAULT[647] : Kistler -KF122 Bewegung mit Weiterschaltung auf Kraft nicht erfolgt, Kraftwert nicht erreicht
   // FAULT[648] : Kistler -KF122 Position liegt ausserhalb der Fahrbereichsgrenze
   // FAULT[649] : Kistler -KF122 Verbindung zum Servoverstärker unterbrochen
   // FAULT[650] : Kistler -KF122 Servoverstärker hat Fehler detektiert / Alarm 650: iSynchro on Setting = 4 OP70.2 / Alarm 650: iSynchro aan Setting = 4 OP70.2
   // FAULT[651] : Kistler -KF122 Kraftüberwachung für Fahrbewegung wurde überschritten / Alarm 651: iSynchro on Result = 4 OP70.2 / Alarm 651: iSynchro aan Result = 4 OP70.2
   // FAULT[652] : Kistler -KF122 Tippbewegung wurde ausserhalb vom Tippbereich angesteuert
   // FAULT[653] : Kistler -KF122 Bewegung mit Stopp auf externes Signal hat kein Stoppsignal erhalten
   // FAULT[654] : Kistler -KF122 Fahrbewegung hat Geschwindigkeit 0 mm/s enthalten
   // FAULT[655] : Kistler -KF122 Umrechnungsfaktor für analogen Ausgang kann nicht gesetzt werden
   // FAULT[656] : Kistler -KF122 Geschwindigkeit Fahrbewegung ausserhalb Grenzen
   // FAULT[657] : Kistler -KF122 Geschwindigkeit Tippbewegung ausserhalb Grenzen
   // FAULT[658] : Kistler -KF122 Bremsentest fehlerhaft
   // FAULT[659] : Kistler -KF122 Unerwarteter Fehler in der Sequenz
   // FAULT[660] : Kistler -KF122 Digitaleingang Timeout
   // FAULT[661] : Kistler -KF122 Sollwertdaten SPS -> maXYmos senden
   // FAULT[662] : Kistler -KF122 Power On fehlt
   // FAULT[663] : Kistler -KF122 Servoantrieb Betriebsbereit fehlt
   // FAULT[664] : Kistler -KF122 Unzulässiges Programm vorgewählt
   // FAULT[665] : Kistler -KF122 Sicherheitsstatus SMES aktiv
   // FAULT[666] : Kistler -KF122 Sicherheitsstatus SMST2 aktiv
   // FAULT[667] : Kistler -KF122 Profinet
   // FAULT[668] : Kistler -KF122 Fehler Servocontroller
   // FAULT[669] : Kistler -KF122 Fehler maXYmos
   // FAULT[670] : Kistler -KF122 Leistung nicht aktiv
   // FAULT[671] : Kistler -KF122 Schutzschalter
   // FAULT[672] : Kistler -KF122 Bremsentest
   // FAULT[673] : Kistler -KF123 Fehler im Setup
   // FAULT[674] : Kistler -KF123 Ungültige Werte für die Sensor X-Kalibrierung
   // FAULT[675] : Kistler -KF123 Ungültige Werte für die Sensor Y-Kalibrierung
   // FAULT[676] : Kistler -KF123 Sensortest war Fehlerhaft
   // FAULT[677] : Kistler -KF123 Eingabe für Kraftbereich Piezo zu klein/gross
   // FAULT[678] : Kistler -KF123 Für Messprogramm wurde kein EO parametriert
   // FAULT[679] : Kistler -KF123 Ein deaktiviertes MP wurde angewählt
   // FAULT[680] : Kistler -KF123 NOK in Folge haben die erlaubte Anzahl überschritten
   // FAULT[681] : Kistler -KF123 Anzahl verpasster Messungen überschritten
   // FAULT[682] : Kistler -KF123 Anzahl der NOK Messungen überschritten
   // FAULT[683] : Kistler -KF123 Hüllkurve Trendüberwachung die Trendgrenze erreicht
   // FAULT[684] : Kistler -KF123 DMS-Sensor nicht angeschlossen oder defekt ist
   // FAULT[685] : Kistler -KF123 Digitalausgang wurde kurz geschlossen
   // FAULT[686] : Kistler -KF123 Sensorversorgung 5 V wird nicht eingehalten
   // FAULT[687] : Kistler -KF123 Speisespannung 24 V wird nicht eingehalten
   // FAULT[688] : Kistler -KF123 Zielverzeichnis hat keinen Speicherplatz
   // FAULT[689] : Kistler -KF123 Zwischenpuffer für unterbrochene Verbindungen voll
   // FAULT[690] : Kistler -KF123 Zugriff auf Variable welche nicht benamt wurde
   // FAULT[691] : Kistler -KF123 Servoverstärker kann keine Leistung hinzugeschaltet werden
   // FAULT[692] : Kistler -KF123 mehrere Fahrbefehle zeitgleich ans Messgerät gesendet
   // FAULT[693] : Kistler -KF123 Sequenz-Element Calculator zwischen MessenStart/Stop plaziert
   // FAULT[694] : Kistler -KF123 Sequenz-Element Calculator sollte durch 0 dividieren
   // FAULT[695] : Kistler -KF123 Bewegung mit Weiterschaltung auf Kraft nicht erfolgt, Kraftwert nicht erreicht
   // FAULT[696] : Kistler -KF123 Position liegt ausserhalb der Fahrbereichsgrenze
   // FAULT[697] : Kistler -KF123 Verbindung zum Servoverstärker unterbrochen
   // FAULT[698] : Kistler -KF123 Servoverstärker hat Fehler detektiert
   // FAULT[699] : Kistler -KF123 Kraftüberwachung für Fahrbewegung wurde überschritten
   // FAULT[700] : Kistler -KF123 Tippbewegung wurde ausserhalb vom Tippbereich angesteuert / Alarm 700: iSynchro on Setting = 4 OP70.3 / Alarm 700: iSynchro aan Setting = 4 OP70.3
   // FAULT[701] : Kistler -KF123 Bewegung mit Stopp auf externes Signal hat kein Stoppsignal erhalten / Alarm 701: iSynchro on Result = 4 OP70.3 / Alarm 701: iSynchro aan Result = 4 OP70.3
   // FAULT[702] : Kistler -KF123 Fahrbewegung hat Geschwindigkeit 0 mm/s enthalten
   // FAULT[703] : Kistler -KF123 Umrechnungsfaktor für analogen Ausgang kann nicht gesetzt werden
   // FAULT[704] : Kistler -KF123 Geschwindigkeit Fahrbewegung ausserhalb Grenzen
   // FAULT[705] : Kistler -KF123 Geschwindigkeit Tippbewegung ausserhalb Grenzen
   // FAULT[706] : Kistler -KF123 Bremsentest fehlerhaft
   // FAULT[707] : Kistler -KF123 Unerwarteter Fehler in der Sequenz
   // FAULT[708] : Kistler -KF123 Digitaleingang Timeout
   // FAULT[709] : Kistler -KF123 Sollwertdaten SPS -> maXYmos senden
   // FAULT[710] : Kistler -KF123 Power On fehlt
   // FAULT[711] : Kistler -KF123 Servoantrieb Betriebsbereit fehlt
   // FAULT[712] : Kistler -KF123 Unzulässiges Programm vorgewählt
   // FAULT[713] : Kistler -KF123 Sicherheitsstatus SMES aktiv
   // FAULT[714] : Kistler -KF123 Sicherheitsstatus SMST2 aktiv
   // FAULT[715] : Kistler -KF123 Profinet
   // FAULT[716] : Kistler -KF123 Fehler Servocontroller
   // FAULT[717] : Kistler -KF123 Fehler maXYmos
   // FAULT[718] : Kistler -KF123 Leistung nicht aktiv
   // FAULT[719] : Kistler -KF123 Schutzschalter
   // FAULT[720] : Kistler -KF123 Bremsentest
   // FAULT[721] : Kistler -KF124 Fehler im Setup
   // FAULT[722] : Kistler -KF124 Ungültige Werte für die Sensor X-Kalibrierung
   // FAULT[723] : Kistler -KF124 Ungültige Werte für die Sensor Y-Kalibrierung
   // FAULT[724] : Kistler -KF124 Sensortest war Fehlerhaft
   // FAULT[725] : Kistler -KF124 Eingabe für Kraftbereich Piezo zu klein/gross
   // FAULT[726] : Kistler -KF124 Für Messprogramm wurde kein EO parametriert
   // FAULT[727] : Kistler -KF124 Ein deaktiviertes MP wurde angewählt
   // FAULT[728] : Kistler -KF124 NOK in Folge haben die erlaubte Anzahl überschritten
   // FAULT[729] : Kistler -KF124 Anzahl verpasster Messungen überschritten
   // FAULT[730] : Kistler -KF124 Anzahl der NOK Messungen überschritten
   // FAULT[731] : Kistler -KF124 Hüllkurve Trendüberwachung die Trendgrenze erreicht
   // FAULT[732] : Kistler -KF124 DMS-Sensor nicht angeschlossen oder defekt ist
   // FAULT[733] : Kistler -KF124 Digitalausgang wurde kurz geschlossen
   // FAULT[734] : Kistler -KF124 Sensorversorgung 5 V wird nicht eingehalten
   // FAULT[735] : Kistler -KF124 Speisespannung 24 V wird nicht eingehalten
   // FAULT[736] : Kistler -KF124 Zielverzeichnis hat keinen Speicherplatz
   // FAULT[737] : Kistler -KF124 Zwischenpuffer für unterbrochene Verbindungen voll
   // FAULT[738] : Kistler -KF124 Zugriff auf Variable welche nicht benamt wurde
   // FAULT[739] : Kistler -KF124 Servoverstärker kann keine Leistung hinzugeschaltet werden
   // FAULT[740] : Kistler -KF124 mehrere Fahrbefehle zeitgleich ans Messgerät gesendet
   // FAULT[741] : Kistler -KF124 Sequenz-Element Calculator zwischen MessenStart/Stop plaziert
   // FAULT[742] : Kistler -KF124 Sequenz-Element Calculator sollte durch 0 dividieren
   // FAULT[743] : Kistler -KF124 Bewegung mit Weiterschaltung auf Kraft nicht erfolgt, Kraftwert nicht erreicht
   // FAULT[744] : Kistler -KF124 Position liegt ausserhalb der Fahrbereichsgrenze
   // FAULT[745] : Kistler -KF124 Verbindung zum Servoverstärker unterbrochen
   // FAULT[746] : Kistler -KF124 Servoverstärker hat Fehler detektiert
   // FAULT[747] : Kistler -KF124 Kraftüberwachung für Fahrbewegung wurde überschritten
   // FAULT[748] : Kistler -KF124 Tippbewegung wurde ausserhalb vom Tippbereich angesteuert
   // FAULT[749] : Kistler -KF124 Bewegung mit Stopp auf externes Signal hat kein Stoppsignal erhalten
   // FAULT[750] : Kistler -KF124 Fahrbewegung hat Geschwindigkeit 0 mm/s enthalten
   // FAULT[751] : Kistler -KF124 Umrechnungsfaktor für analogen Ausgang kann nicht gesetzt werden
   // FAULT[752] : Kistler -KF124 Geschwindigkeit Fahrbewegung ausserhalb Grenzen
   // FAULT[753] : Kistler -KF124 Geschwindigkeit Tippbewegung ausserhalb Grenzen
   // FAULT[754] : Kistler -KF124 Bremsentest fehlerhaft
   // FAULT[755] : Kistler -KF124 Unerwarteter Fehler in der Sequenz
   // FAULT[756] : Kistler -KF124 Digitaleingang Timeout
   // FAULT[757] : Kistler -KF124 Sollwertdaten SPS -> maXYmos senden
   // FAULT[758] : Kistler -KF124 Power On fehlt
   // FAULT[759] : Kistler -KF124 Servoantrieb Betriebsbereit fehlt
   // FAULT[760] : Kistler -KF124 Unzulässiges Programm vorgewählt
   // FAULT[761] : Kistler -KF124 Sicherheitsstatus SMES aktiv
   // FAULT[762] : Kistler -KF124 Sicherheitsstatus SMST2 aktiv
   // FAULT[763] : Kistler -KF124 Profinet
   // FAULT[764] : Kistler -KF124 Fehler Servocontroller
   // FAULT[765] : Kistler -KF124 Fehler maXYmos
   // FAULT[766] : Kistler -KF124 Leistung nicht aktiv
   // FAULT[767] : Kistler -KF124 Schutzschalter
   // FAULT[768] : Kistler -KF124 Bremsentest
   // FAULT[769] : Kistler -KF125 Fehler im Setup
   // FAULT[770] : Kistler -KF125 Ungültige Werte für die Sensor X-Kalibrierung
   // FAULT[771] : Kistler -KF125 Ungültige Werte für die Sensor Y-Kalibrierung
   // FAULT[772] : Kistler -KF125 Sensortest war Fehlerhaft
   // FAULT[773] : Kistler -KF125 Eingabe für Kraftbereich Piezo zu klein/gross
   // FAULT[774] : Kistler -KF125 Für Messprogramm wurde kein EO parametriert
   // FAULT[775] : Kistler -KF125 Ein deaktiviertes MP wurde angewählt
   // FAULT[776] : Kistler -KF125 NOK in Folge haben die erlaubte Anzahl überschritten
   // FAULT[777] : Kistler -KF125 Anzahl verpasster Messungen überschritten
   // FAULT[778] : Kistler -KF125 Anzahl der NOK Messungen überschritten
   // FAULT[779] : Kistler -KF125 Hüllkurve Trendüberwachung die Trendgrenze erreicht
   // FAULT[780] : Kistler -KF125 DMS-Sensor nicht angeschlossen oder defekt ist
   // FAULT[781] : Kistler -KF125 Digitalausgang wurde kurz geschlossen
   // FAULT[782] : Kistler -KF125 Sensorversorgung 5 V wird nicht eingehalten
   // FAULT[783] : Kistler -KF125 Speisespannung 24 V wird nicht eingehalten
   // FAULT[784] : Kistler -KF125 Zielverzeichnis hat keinen Speicherplatz
   // FAULT[785] : Kistler -KF125 Zwischenpuffer für unterbrochene Verbindungen voll
   // FAULT[786] : Kistler -KF125 Zugriff auf Variable welche nicht benamt wurde
   // FAULT[787] : Kistler -KF125 Servoverstärker kann keine Leistung hinzugeschaltet werden
   // FAULT[788] : Kistler -KF125 mehrere Fahrbefehle zeitgleich ans Messgerät gesendet
   // FAULT[789] : Kistler -KF125 Sequenz-Element Calculator zwischen MessenStart/Stop plaziert
   // FAULT[790] : Kistler -KF125 Sequenz-Element Calculator sollte durch 0 dividieren
   // FAULT[791] : Kistler -KF125 Bewegung mit Weiterschaltung auf Kraft nicht erfolgt, Kraftwert nicht erreicht
   // FAULT[792] : Kistler -KF125 Position liegt ausserhalb der Fahrbereichsgrenze
   // FAULT[793] : Kistler -KF125 Verbindung zum Servoverstärker unterbrochen
   // FAULT[794] : Kistler -KF125 Servoverstärker hat Fehler detektiert
   // FAULT[795] : Kistler -KF125 Kraftüberwachung für Fahrbewegung wurde überschritten
   // FAULT[796] : Kistler -KF125 Tippbewegung wurde ausserhalb vom Tippbereich angesteuert
   // FAULT[797] : Kistler -KF125 Bewegung mit Stopp auf externes Signal hat kein Stoppsignal erhalten
   // FAULT[798] : Kistler -KF125 Fahrbewegung hat Geschwindigkeit 0 mm/s enthalten
   // FAULT[799] : Kistler -KF125 Umrechnungsfaktor für analogen Ausgang kann nicht gesetzt werden
   // FAULT[800] : Kistler -KF125 Geschwindigkeit Fahrbewegung ausserhalb Grenzen / Alarm 800: Camera - Component not detected_OP70_2 / Alarm 800: Camera - Component niet gedetecteerd_OP70_2
   // FAULT[801] : Kistler -KF125 Geschwindigkeit Tippbewegung ausserhalb Grenzen
   // FAULT[802] : Kistler -KF125 Bremsentest fehlerhaft
   // FAULT[803] : Kistler -KF125 Unerwarteter Fehler in der Sequenz
   // FAULT[804] : Kistler -KF125 Digitaleingang Timeout
   // FAULT[805] : Kistler -KF125 Sollwertdaten SPS -> maXYmos senden
   // FAULT[806] : Kistler -KF125 Power On fehlt
   // FAULT[807] : Kistler -KF125 Servoantrieb Betriebsbereit fehlt
   // FAULT[808] : Kistler -KF125 Unzulässiges Programm vorgewählt
   // FAULT[809] : Kistler -KF125 Sicherheitsstatus SMES aktiv
   // FAULT[810] : Kistler -KF125 Sicherheitsstatus SMST2 aktiv
   // FAULT[811] : Kistler -KF125 Profinet
   // FAULT[812] : Kistler -KF125 Fehler Servocontroller
   // FAULT[813] : Kistler -KF125 Fehler maXYmos
   // FAULT[814] : Kistler -KF125 Leistung nicht aktiv
   // FAULT[815] : Kistler -KF125 Schutzschalter
   // FAULT[816] : Kistler -KF125 Bremsentest
   // FAULT[817] : Kistler -KF126 Fehler im Setup
   // FAULT[818] : Kistler -KF126 Ungültige Werte für die Sensor X-Kalibrierung
   // FAULT[819] : Kistler -KF126 Ungültige Werte für die Sensor Y-Kalibrierung
   // FAULT[820] : Kistler -KF126 Sensortest war Fehlerhaft
   // FAULT[821] : Kistler -KF126 Eingabe für Kraftbereich Piezo zu klein/gross
   // FAULT[822] : Kistler -KF126 Für Messprogramm wurde kein EO parametriert
   // FAULT[823] : Kistler -KF126 Ein deaktiviertes MP wurde angewählt
   // FAULT[824] : Kistler -KF126 NOK in Folge haben die erlaubte Anzahl überschritten
   // FAULT[825] : Kistler -KF126 Anzahl verpasster Messungen überschritten
   // FAULT[826] : Kistler -KF126 Anzahl der NOK Messungen überschritten
   // FAULT[827] : Kistler -KF126 Hüllkurve Trendüberwachung die Trendgrenze erreicht
   // FAULT[828] : Kistler -KF126 DMS-Sensor nicht angeschlossen oder defekt ist
   // FAULT[829] : Kistler -KF126 Digitalausgang wurde kurz geschlossen
   // FAULT[830] : Kistler -KF126 Sensorversorgung 5 V wird nicht eingehalten
   // FAULT[831] : Kistler -KF126 Speisespannung 24 V wird nicht eingehalten
   // FAULT[832] : Kistler -KF126 Zielverzeichnis hat keinen Speicherplatz
   // FAULT[833] : Kistler -KF126 Zwischenpuffer für unterbrochene Verbindungen voll
   // FAULT[834] : Kistler -KF126 Zugriff auf Variable welche nicht benamt wurde
   // FAULT[835] : Kistler -KF126 Servoverstärker kann keine Leistung hinzugeschaltet werden
   // FAULT[836] : Kistler -KF126 mehrere Fahrbefehle zeitgleich ans Messgerät gesendet
   // FAULT[837] : Kistler -KF126 Sequenz-Element Calculator zwischen MessenStart/Stop plaziert
   // FAULT[838] : Kistler -KF126 Sequenz-Element Calculator sollte durch 0 dividieren
   // FAULT[839] : Kistler -KF126 Bewegung mit Weiterschaltung auf Kraft nicht erfolgt, Kraftwert nicht erreicht
   // FAULT[840] : Kistler -KF126 Position liegt ausserhalb der Fahrbereichsgrenze
   // FAULT[841] : Kistler -KF126 Verbindung zum Servoverstärker unterbrochen
   // FAULT[842] : Kistler -KF126 Servoverstärker hat Fehler detektiert
   // FAULT[843] : Kistler -KF126 Kraftüberwachung für Fahrbewegung wurde überschritten
   // FAULT[844] : Kistler -KF126 Tippbewegung wurde ausserhalb vom Tippbereich angesteuert
   // FAULT[845] : Kistler -KF126 Bewegung mit Stopp auf externes Signal hat kein Stoppsignal erhalten
   // FAULT[846] : Kistler -KF126 Fahrbewegung hat Geschwindigkeit 0 mm/s enthalten
   // FAULT[847] : Kistler -KF126 Umrechnungsfaktor für analogen Ausgang kann nicht gesetzt werden
   // FAULT[848] : Kistler -KF126 Geschwindigkeit Fahrbewegung ausserhalb Grenzen
   // FAULT[849] : Kistler -KF126 Geschwindigkeit Tippbewegung ausserhalb Grenzen
   // FAULT[850] : Kistler -KF126 Bremsentest fehlerhaft
   // FAULT[851] : Kistler -KF126 Unerwarteter Fehler in der Sequenz
   // FAULT[852] : Kistler -KF126 Digitaleingang Timeout
   // FAULT[853] : Kistler -KF126 Sollwertdaten SPS -> maXYmos senden
   // FAULT[854] : Kistler -KF126 Power On fehlt
   // FAULT[855] : Kistler -KF126 Servoantrieb Betriebsbereit fehlt
   // FAULT[856] : Kistler -KF126 Unzulässiges Programm vorgewählt
   // FAULT[857] : Kistler -KF126 Sicherheitsstatus SMES aktiv
   // FAULT[858] : Kistler -KF126 Sicherheitsstatus SMST2 aktiv
   // FAULT[859] : Kistler -KF126 Profinet
   // FAULT[860] : Kistler -KF126 Fehler Servocontroller
   // FAULT[861] : Kistler -KF126 Fehler maXYmos
   // FAULT[862] : Kistler -KF126 Leistung nicht aktiv
   // FAULT[863] : Kistler -KF126 Schutzschalter
   // FAULT[864] : Kistler -KF126 Bremsentest
   // FAULT[865] : Kein Hülse in Zustellung
   // FAULT[866] : Kein Hülse in Ablage
   // FAULT[867] : Cognex Scanner -BX200 Fehler
   // FAULT[868] : Cognex Scanner -BX200 Fehler Timeout
   // FAULT[869] : fehler869
   // FAULT[870] : fehler870
   // FAULT[871] : fehler871
   // FAULT[872] : fehler872
   // FAULT[873] : Cognex Kamera -BXxxx Spiegelung PID n.i.O.
   // FAULT[874] : Cognex Kamera -BXxxx Programmnummer ungültig
   // FAULT[875] : Cognex Kamera -BXxxx Beleuchtungscheck n.i.O.
   // FAULT[876] : Cognex Kamera -BXxxx Fehler Offline
   // FAULT[877] : Cognex Kamera -BXxxx Ablauffehler
   // FAULT[878] : Cognex Kamera -BXxxx Fehler
   // FAULT[879] : Cognex Kamera -BXxxx Fehler Timeout
   // FAULT[880] : fehler880
   // FAULT[881] : fehler881
   // FAULT[882] : fehler882
   // FAULT[883] : fehler883
   // FAULT[884] : fehler884
   // FAULT[885] : fehler885
   // FAULT[886] : fehler886
   // FAULT[887] : fehler887
   // FAULT[888] : fehler888
   // FAULT[889] : fehler889
   // FAULT[890] : fehler890
   // FAULT[891] : fehler891
   // FAULT[892] : fehler892
   // FAULT[893] : fehler893
   // FAULT[894] : fehler894
   // FAULT[895] : fehler895
   // FAULT[896] : fehler896
   // FAULT[897] : fehler897
   // FAULT[898] : fehler898
   // FAULT[899] : fehler899
   // FAULT[900] : fehler900
   // FAULT[901] : fehler901
   // FAULT[902] : fehler902
   // FAULT[903] : fehler903
   // FAULT[904] : fehler904
   // FAULT[905] : fehler905
   // FAULT[906] : fehler906
   // FAULT[907] : fehler907
   // FAULT[908] : fehler908
   // FAULT[909] : fehler909
   // FAULT[910] : fehler910
   // FAULT[911] : fehler911
   // FAULT[912] : fehler912
   // FAULT[913] : fehler913
   // FAULT[914] : fehler914
   // FAULT[915] : fehler915
   // FAULT[916] : fehler916
   // FAULT[917] : fehler917
   // FAULT[918] : fehler918
   // FAULT[919] : fehler919
   // FAULT[920] : fehler920
   // FAULT[921] : fehler921
   // FAULT[922] : fehler922
   // FAULT[923] : fehler923
   // FAULT[924] : fehler924
   // FAULT[925] : fehler925
   // FAULT[926] : fehler926
   // FAULT[927] : fehler927
   // FAULT[928] : fehler928
   // FAULT[929] : fehler929
   // FAULT[930] : fehler930
   // FAULT[931] : fehler931
   // FAULT[932] : fehler932
   // FAULT[933] : fehler933
   // FAULT[934] : fehler934
   // FAULT[935] : fehler935
   // FAULT[936] : fehler936
   // FAULT[937] : fehler937
   // FAULT[938] : fehler938
   // FAULT[939] : fehler939
   // FAULT[940] : fehler940
   // FAULT[941] : fehler941
   // FAULT[942] : fehler942
   // FAULT[943] : fehler943
   // FAULT[944] : fehler944
   // FAULT[945] : fehler945
   // FAULT[946] : fehler946
   // FAULT[947] : fehler947
   // FAULT[948] : fehler948
   // FAULT[949] : fehler949
   // FAULT[950] : fehler950
   // FAULT[951] : fehler951
   // FAULT[952] : fehler952
   // FAULT[953] : fehler953
   // FAULT[954] : fehler954
   // FAULT[955] : fehler955
   // FAULT[956] : fehler956
   // FAULT[957] : fehler957
   // FAULT[958] : fehler958
   // FAULT[959] : fehler959
   // FAULT[960] : fehler960
   // FAULT[961] : fehler961
   // FAULT[962] : fehler962
   // FAULT[963] : fehler963
   // FAULT[964] : fehler964
   // FAULT[965] : fehler965
   // FAULT[966] : fehler966
   // FAULT[967] : fehler967
   // FAULT[968] : fehler968
   // FAULT[969] : fehler969
   // FAULT[970] : fehler970
   // FAULT[971] : fehler971
   // FAULT[972] : fehler972
   // FAULT[973] : fehler973
   // FAULT[974] : fehler974
   // FAULT[975] : fehler975
   // FAULT[976] : fehler976
   // FAULT[977] : fehler977
   // FAULT[978] : fehler978
   // FAULT[979] : fehler979
   // FAULT[980] : fehler980
   // FAULT[981] : fehler981
   // FAULT[982] : fehler982
   // FAULT[983] : fehler983
   // FAULT[984] : fehler984
   // FAULT[985] : fehler985
   // FAULT[986] : fehler986
   // FAULT[987] : fehler987
   // FAULT[988] : fehler988
   // FAULT[989] : fehler989
   // FAULT[990] : fehler990
   // FAULT[991] : fehler991
   // FAULT[992] : fehler992
   // FAULT[993] : fehler993
   // FAULT[994] : fehler994
   // FAULT[995] : fehler995
   // FAULT[996] : fehler996
   // FAULT[997] : fehler997
   // FAULT[998] : fehler998
   // FAULT[999] : fehler999
   // FAULT[1000] : fehler1000
   // FAULT[1001] : fehler1001
   // FAULT[1002] : fehler1002
   // FAULT[1003] : fehler1003
   // FAULT[1004] : fehler1004
   // FAULT[1005] : fehler1005
   // FAULT[1006] : fehler1006
   // FAULT[1007] : fehler1007
   // FAULT[1008] : fehler1008
   // FAULT[1009] : fehler1009
   // FAULT[1010] : fehler1010
   // FAULT[1011] : fehler1011
   // FAULT[1012] : fehler1012
   // FAULT[1013] : fehler1013
   // FAULT[1014] : fehler1014
   // FAULT[1015] : fehler1015
   // FAULT[1016] : fehler1016
   // FAULT[1017] : fehler1017
   // FAULT[1018] : fehler1018
   // FAULT[1019] : fehler1019
   // FAULT[1020] : fehler1020
   // FAULT[1021] : fehler1021
   // FAULT[1022] : fehler1022
   // FAULT[1023] : fehler1023
   // FAULT[1024] : fehler1024
   // WARNING[1] : Allg: kein Text
   // WARNING[2] : Allg: kein Text
   // WARNING[3] : Allg: keine Betriebsart aktiv / General Warning: No operating mode active(Hand/Auto) / Algemene waarschuwing: geen bedrijfsmodus actief (hand/auto)
   // WARNING[4] : Allg: Betriebsart Einzelschritt / General Warning: Single step mode / Algemene waarschuwing: één staps modus actief
   // WARNING[5] : Allg: Betriebsart Service / General Warning: Service mode / Algemene waarschuwing: servicemodus
   // WARNING[6] : Allg: Typwechsel aktiv / General Warning: Type change active / Algemene waarschuwing: Typewijziging actief
   // WARNING[7] : Allg: kein Text
   // WARNING[8] : Allg: kein Text
   // WARNING[9] : Allg: Anforderung Schutzgitter Station öffnen / General Warning: Safety Door 1 opened / Algemene waarschuwing: veiligheidsdeur 1 geopend
   // WARNING[10] : Allg: Anforderung Schutzgitter Drucker öffnen
   // WARNING[11] : Allg: Anforderung Schutzgitter öffnen
   // WARNING[12] : Allg: kein Text
   // WARNING[13] : Allg: kein Text
   // WARNING[14] : Allg: kein Text
   // WARNING[15] : Allg: kein Text
   // WARNING[16] : Allg: Schutztürüberbrückung Station ("E2") aktiv
   // WARNING[17] : Allg: kein Text
   // WARNING[18] : Allg: kein Text
   // WARNING[19] : Allg: kein Text
   // WARNING[20] : EKS: kein Key vorhanden [+ZP-SH01] / EKS: No key available[+ZP01-271SH01] / EKS: Geen sleutel beschikbaar[+ZP01-271SH01]
   // WARNING[21] : EKS: Ablaufdatum "" überschritten [+ZP-SH01] / EKS: Expiration date exceeded[+ZP01-271SH01] / EKS: Vervaldatum overschreden[+ZP01-271SH01]
   // WARNING[22] : EKS: Kostenstelle n.i.O. [+ZP-SH01] / EKS: Cost Center NOK[+ZP01-271SH01] / EKS: Kostenplaats NOK[+ZP01-271SH01]
   // WARNING[23] : EKS: Berechtigung n.i.O. [+ZP-SH01] / EKS: Authorization NOK[+ZP01-271SH01] / EKS: Autorisatie NOK[+ZP01-271SH01]
   // WARNING[24] : EKS: Läuft am "" ab [+ZP-SH01] / EKS: Expires on[+ZP01-271SH01] / EKS: Verloopt op[+ZP01-271SH01]
   // WARNING[25] : Allg: kein Text
   // WARNING[26] : Allg: kein Text
   // WARNING[27] : Allg: kein Text
   // WARNING[28] : Allg: kein Text
   // WARNING[29] : Allg: kein Text
   // WARNING[30] : Allg: kein Text
   // WARNING[31] : Allg: kein Text
   // WARNING[32] : Allg: kein Text
   // WARNING[33] : Allg: Meldung Profinet/Ehternet Scalance n.i.O.[+S01-275XF1] / General: Message Profinet / Ehternet Scalance NOK [+S01-275XF1] / Algemeen: Bericht Profinet / Ehternet Scalance NOK [+S01-275XF1]
   // WARNING[34] : Allg: Schaltschrank Temperatur n.i.O. [i0. 7] / General: Control cabinet temperature NIO [+S01- BG0.7] / Algemeen: Schakelkasttemperatuur NIO [+S01- BG0.7]
   // WARNING[35] : Allg: Kühlgerät Zustand n.i.O. [+S01-EC01]
   // WARNING[36] : Allg: kein Text
   // WARNING[37] : Allg: kein Text
   // WARNING[38] : Allg: kein Text
   // WARNING[39] : Allg: kein Text
   // WARNING[40] : Allg: kein Text
   // WARNING[41] : <Zentralschmierung>: Füllstand "min" [+M01-BL3.7]
   // WARNING[42] : <Zentralschmierung>: Druck nicht erreicht [+M01-BP50.6]
   // WARNING[43] : Allg: kein Text
   // WARNING[44] : Allg: kein Text
   // WARNING[45] : Allg: kein Text
   // WARNING[46] : Allg: kein Text
   // WARNING[47] : Allg: kein Text
   // WARNING[48] : Allg: kein Text
   // WARNING[49] : Allg: kein Text
   // WARNING[50] : Allg: Mindestens eine Bearbeitung abgewählt / General: Removed at least one processing. / Algemeen: Minstens één verwerking verwijderd.
   // WARNING[51] : Allg: Stau im Auslauf Station / General: Congestion at Out of Station / Algemeen: congestie bij buiten het station
   // WARNING[52] : Allg: kein Text
   // WARNING[53] : Allg: kein Text
   // WARNING[54] : Allg: kein Text
   // WARNING[55] : Allg: kein Text
   // WARNING[56] : Allg: kein Text
   // WARNING[57] : Allg: kein Text
   // WARNING[58] : Allg: kein Text
   // WARNING[59] : Allg: kein Text
   // WARNING[60] : Allg: kein Text
   // WARNING[61] : Allg: kein Text
   // WARNING[62] : Allg: kein Text
   // WARNING[63] : Allg: kein Text
   // WARNING[64] : Allg: kein Text
   // WARNING[65] : Allg: kein Text
   // WARNING[66] : Allg: kein Text
   // WARNING[67] : Allg: kein Text
   // WARNING[68] : Allg: kein Text
   // WARNING[69] : Allg: kein Text
   // WARNING[70] : Allg: kein Text
   // WARNING[71] : Allg: kein Text
   // WARNING[72] : Allg: kein Text
   // WARNING[73] : Allg: kein Text
   // WARNING[74] : Allg: kein Text
   // WARNING[75] : Allg: kein Text
   // WARNING[76] : Allg: kein Text
   // WARNING[77] : Allg: kein Text
   // WARNING[78] : Allg: kein Text
   // WARNING[79] : Allg: kein Text
   // WARNING[80] : Zentrale: Verbindung zur zentralen Verkettung gestört
   // WARNING[81] : Zentrale: Zentral Maschine Aus von VK angefordert
   // WARNING[82] : Zentrale: Bahnantriebe nicht eingeschaltet
   // WARNING[83] : Zentrale: Bahnantriebe nicht eingeschaltet
   // WARNING[84] : Zentrale: Abgewählt
   // WARNING[85] : Zentrale: kein Text
   // WARNING[86] : Zentrale: kein Text
   // WARNING[87] : Zentrale: kein Text
   // WARNING[88] : Zentrale: kein Text
   // WARNING[89] : Zentrale: kein Text
   // WARNING[90] : Ethernet: Fehler Daten senden
   // WARNING[91] : Ethernet: Fehler Daten empfangen
   // WARNING[92] : Ethernet: kein Text
   // WARNING[93] : Ethernet: kein Text
   // WARNING[94] : Ethernet: kein Text
   // WARNING[95] : Ethernet: kein Text
   // WARNING[96] : BDE: Keine Verbindung zum BDE-System (Taktzeit)
   // WARNING[97] : BDE: Keine Verbindung zum BDE-System (Stückzahl)
   // WARNING[98] : BDE: Keine Verbindung zum BDE-System (Maschinenzustand)
   // WARNING[99] : BDE: Keine Verbindung zum BDE-System (Meldung)
   // WARNING[100] : Allg: kein Text
   // WARNING[101] : Allg: kein Text
   // WARNING[102] : Allg: kein Text
   // WARNING[103] : Allg: kein Text
   // WARNING[104] : Allg: kein Text
   // WARNING[105] : Allg: kein Text
   // WARNING[106] : Allg: kein Text
   // WARNING[107] : Allg: kein Text
   // WARNING[108] : Allg: kein Text
   // WARNING[109] : Allg: kein Text
   // WARNING[110] : Teilemangel: Station leer / Part controle: Station Empty / Onderdeelcontrole: Station Leeg
   // WARNING[111] : Teilemangel: kein Text
   // WARNING[112] : Teilemangel: kein Text
   // WARNING[113] : Teilemangel: kein Text
   // WARNING[114] : Teilemangel: kein Text
   // WARNING[115] : Teilemangel: kein Text
   // WARNING[116] : Teilemangel: kein Text
   // WARNING[117] : Teilemangel: kein Text
   // WARNING[118] : Teilemangel: kein Text
   // WARNING[119] : Allg: kein Text
   // WARNING[120] : Allg: kein Text
   // WARNING[121] : Allg: kein Text
   // WARNING[122] : Allg: kein Text
   // WARNING[123] : Allg: kein Text
   // WARNING[124] : Allg: kein Text
   // WARNING[125] : Allg: kein Text
   // WARNING[126] : Allg: kein Text
   // WARNING[127] : Allg: kein Text
   // WARNING[128] : Allg: kein Text
   // WARNING[129] : Allg: kein Text
   // WARNING[130] : Allg: kein Text
   // WARNING[131] : Allg: kein Text
   // WARNING[132] : Allg: kein Text
   // WARNING[133] : Allg: kein Text
   // WARNING[134] : Allg: kein Text
   // WARNING[135] : Allg: kein Text
   // WARNING[136] : Allg: kein Text
   // WARNING[137] : Allg: kein Text
   // WARNING[138] : Allg: kein Text
   // WARNING[139] : Allg: kein Text
   // WARNING[140] : Allg: kein Text
   // WARNING[141] : Allg: kein Text
   // WARNING[142] : Allg: kein Text
   // WARNING[143] : Allg: kein Text
   // WARNING[144] : Allg: kein Text
   // WARNING[145] : Allg: kein Text
   // WARNING[146] : Allg: kein Text
   // WARNING[147] : Allg: kein Text
   // WARNING[148] : Allg: kein Text
   // WARNING[149] : Allg: kein Text
   // WARNING[150] : Allg: kein Text
   // WARNING[151] : Allg: kein Text
   // WARNING[152] : Allg: kein Text
   // WARNING[153] : Allg: kein Text
   // WARNING[154] : Allg: kein Text
   // WARNING[155] : Allg: kein Text
   // WARNING[156] : Allg: kein Text
   // WARNING[157] : Allg: kein Text
   // WARNING[158] : Allg: kein Text
   // WARNING[159] : Allg: kein Text
   // WARNING[160] : Allg: kein Text
   // WARNING[161] : warning161
   // WARNING[162] : warning162
   // WARNING[163] : warning163
   // WARNING[164] : warning164
   // WARNING[165] : warning165
   // WARNING[166] : warning166
   // WARNING[167] : warning167
   // WARNING[168] : warning168
   // WARNING[169] : warning169
   // WARNING[170] : warning170
   // WARNING[171] : warning171
   // WARNING[172] : warning172
   // WARNING[173] : warning173
   // WARNING[174] : warning174
   // WARNING[175] : warning175
   // WARNING[176] : warning176
   // WARNING[177] : warning177
   // WARNING[178] : warning178
   // WARNING[179] : warning179
   // WARNING[180] : warning180
   // WARNING[181] : warning181
   // WARNING[182] : warning182
   // WARNING[183] : warning183
   // WARNING[184] : warning184
   // WARNING[185] : warning185
   // WARNING[186] : warning186
   // WARNING[187] : warning187
   // WARNING[188] : warning188
   // WARNING[189] : warning189
   // WARNING[190] : warning190 / Warning 190: Feeder Unit Empty Damper Cap [+M01- BG55.4] / Waarschuwing 190: Automatische aanvoerunit van de demper cap is leeg [+M01- BG55.4]
   // WARNING[191] : warning191 / Warning 191: Feeder Unit Empty Ball [+M01- BG56.0] / Waarschuwing 191: Automatische aanvoerunit van de bal is leeg[+M01- BG56.0]
   // WARNING[192] : warning192 / Warning 192: Feeder Unit Empty Screw [+M01- BG56.1] / Waarschuwing 192: Automatische aanvoerunit van de schroeven is leeg [+M01- BG56.1]
   // WARNING[193] : warning193
   // WARNING[194] : warning194
   // WARNING[195] : warning195
   // WARNING[196] : warning196
   // WARNING[197] : warning197
   // WARNING[198] : warning198
   // WARNING[199] : warning199
   // WARNING[200] : warning200
   // WARNING[201] : Schrauber mPro Systemwarnung [+S01-KF100]
   // WARNING[202] : warning202
   // WARNING[203] : warning203
   // WARNING[204] : warning204
   // WARNING[205] : warning205
   // WARNING[206] : warning206
   // WARNING[207] : warning207
   // WARNING[208] : warning208
   // WARNING[209] : warning209
   // WARNING[210] : warning210
   // WARNING[211] : warning211
   // WARNING[212] : warning212
   // WARNING[213] : warning213
   // WARNING[214] : warning214
   // WARNING[215] : warning215
   // WARNING[216] : warning216
   // WARNING[217] : warning217
   // WARNING[218] : warning218
   // WARNING[219] : warning219
   // WARNING[220] : warning220
   // WARNING[221] : warning221
   // WARNING[222] : warning222
   // WARNING[223] : warning223
   // WARNING[224] : warning224
   // WARNING[225] : warning225
   // WARNING[226] : warning226
   // WARNING[227] : warning227
   // WARNING[228] : warning228
   // WARNING[229] : warning229
   // WARNING[230] : warning230
   // WARNING[231] : warning231
   // WARNING[232] : warning232
   // WARNING[233] : warning233
   // WARNING[234] : warning234
   // WARNING[235] : warning235
   // WARNING[236] : warning236
   // WARNING[237] : warning237
   // WARNING[238] : warning238
   // WARNING[239] : warning239
   // WARNING[240] : warning240
   // WARNING[241] : warning241
   // WARNING[242] : warning242
   // WARNING[243] : warning243
   // WARNING[244] : warning244
   // WARNING[245] : warning245
   // WARNING[246] : warning246
   // WARNING[247] : warning247
   // WARNING[248] : warning248
   // WARNING[249] : warning249
   // WARNING[250] : warning250
   // WARNING[251] : warning251
   // WARNING[252] : warning252
   // WARNING[253] : warning253
   // WARNING[254] : warning254
   // WARNING[255] : warning255
   // WARNING[256] : warning256
   // WARNING[257] : Roboter 1 - nicht in Automatik
   // WARNING[258] : Roboter 1 - Bremsentest wird angefordert
   // WARNING[259] : Roboter 1 - Bremsentest Monitoringzeit wurde überschritten
   // WARNING[260] : Roboter 1 - Bremsentest wird durchgeführt
   // WARNING[261] : Roboter 1 - Bremse ist defekt
   // WARNING[262] : Roboter 1 - Bremse hat Verschleissgrenze erreicht
   // WARNING[263] : Roboter 1 - nicht referenziert
   // WARNING[264] : Roboter 1 - Justagefehler
   // WARNING[265] : warning265
   // WARNING[266] : warning266
   // WARNING[267] : warning267
   // WARNING[268] : warning268
   // WARNING[269] : warning269
   // WARNING[270] : warning270
   // WARNING[271] : warning271
   // WARNING[272] : warning272
   // WARNING[273] : Roboter 2 - nicht in Automatik
   // WARNING[274] : Roboter 2 - Bremsentest wird angefordert
   // WARNING[275] : Roboter 2 - Monitoringzeit wurde überschritten
   // WARNING[276] : Roboter 2 - Bremsentest wird durchgeführt
   // WARNING[277] : Roboter 2 - Bremse ist defekt
   // WARNING[278] : Roboter 2 - Bremse hat Verschleissgrenze erreicht
   // WARNING[279] : Roboter 2 - nicht referenziert
   // WARNING[280] : Roboter 2 - Justagefehler
   // WARNING[281] : warning281
   // WARNING[282] : warning282
   // WARNING[283] : warning283
   // WARNING[284] : warning284
   // WARNING[285] : warning285
   // WARNING[286] : warning286
   // WARNING[287] : warning287
   // WARNING[288] : warning288
   // WARNING[289] : warning289
   // WARNING[290] : warning290
   // WARNING[291] : warning291
   // WARNING[292] : warning292
   // WARNING[293] : warning293
   // WARNING[294] : warning294
   // WARNING[295] : warning295
   // WARNING[296] : warning296
   // WARNING[297] : warning297
   // WARNING[298] : warning298
   // WARNING[299] : warning299
   // WARNING[300] : warning300 / Warning 300:: X1- The assumed level of NOK has been reached / Waarschuwing 300: X1- Het veronderstelde niveau van NOK is bereikt
   // WARNING[301] : warning301 / Warning 301: MES interlock is OFF, on this machine / Waarschuwing 301: MES-interlock is uitgeschakeld op deze machine
   // WARNING[302] : warning302 / Warning 302: MES Traceability is OFF, on this machine / Waarschuwing 302: MES-Traceerbaarheid is uitgeschakeld op deze machine
   // WARNING[303] : warning303 / Waarschuwing 303: Wachten op MES antwoord (iSynchro=2) / Warning 303: Waiting for MES response (iSynchro = 2)
   // WARNING[304] : warning304 / Warning 304: MES switched to OFF : reason Golden part / Waarschuwing 304: MES uitgeschakeld : reden Golden Part
   // WARNING[305] : warning305 / Warning 305: MES switched to OFF : reason Maintenance / Waarschuwing 305: MES uitgeschakeld : reden Maintenance
   // WARNING[306] : warning306 / Warning 306: MES switched to OFF : reason MSA / Waarschuwing 306: MES uitgeschakeld : reden MSA
   // WARNING[307] : warning307 / Warning 307: MES switched to OFF : reason Test purposes / Waarschuwing 307: MES uitgeschakeld : reden Test Purposes
   // WARNING[308] : warning308
   // WARNING[309] : warning309
   // WARNING[310] : warning310
   // WARNING[311] : warning311
   // WARNING[312] : warning312
   // WARNING[313] : warning313
   // WARNING[314] : warning314
   // WARNING[315] : warning315
   // WARNING[316] : warning316
   // WARNING[317] : warning317
   // WARNING[318] : warning318
   // WARNING[319] : warning319
   // WARNING[320] : warning320
   // WARNING[321] : Achse: Vertikalschlitten - Warnung [+S01-KF110]
   // WARNING[322] : Achse: Vertikalschlitten - Anforderung Bremsentest [+S01-KF110]
   // WARNING[323] : Achse: Vertikalschlitten - Override nicht 100%
   // WARNING[324] : warning324
   // WARNING[325] : warning325
   // WARNING[326] : warning326
   // WARNING[327] : Achse: MA10 Test Stop ist aktiv
   // WARNING[328] : warning328
   // WARNING[329] : warning329
   // WARNING[330] : warning330
   // WARNING[331] : warning331
   // WARNING[332] : warning332
   // WARNING[333] : warning333
   // WARNING[334] : warning334
   // WARNING[335] : warning335
   // WARNING[336] : warning336
   // WARNING[337] : warning337
   // WARNING[338] : warning338
   // WARNING[339] : warning339
   // WARNING[340] : warning340
   // WARNING[341] : warning341
   // WARNING[342] : warning342
   // WARNING[343] : warning343
   // WARNING[344] : warning344
   // WARNING[345] : warning345
   // WARNING[346] : warning346
   // WARNING[347] : warning347
   // WARNING[348] : warning348
   // WARNING[349] : warning349
   // WARNING[350] : warning350
   // WARNING[351] : warning351
   // WARNING[352] : warning352
   // WARNING[353] : warning353
   // WARNING[354] : warning354
   // WARNING[355] : warning355
   // WARNING[356] : warning356
   // WARNING[357] : warning357
   // WARNING[358] : warning358
   // WARNING[359] : warning359
   // WARNING[360] : warning360
   // WARNING[361] : warning361
   // WARNING[362] : warning362
   // WARNING[363] : warning363
   // WARNING[364] : warning364
   // WARNING[365] : warning365
   // WARNING[366] : warning366
   // WARNING[367] : warning367
   // WARNING[368] : warning368
   // WARNING[369] : warning369
   // WARNING[370] : warning370
   // WARNING[371] : warning371
   // WARNING[372] : warning372
   // WARNING[373] : warning373
   // WARNING[374] : warning374
   // WARNING[375] : warning375
   // WARNING[376] : warning376
   // WARNING[377] : warning377
   // WARNING[378] : warning378
   // WARNING[379] : warning379
   // WARNING[380] : warning380
   // WARNING[381] : warning381
   // WARNING[382] : warning382
   // WARNING[383] : warning383
   // WARNING[384] : warning384
   // WARNING[385] : warning385
   // WARNING[386] : warning386
   // WARNING[387] : warning387
   // WARNING[388] : warning388
   // WARNING[389] : warning389
   // WARNING[390] : warning390
   // WARNING[391] : warning391
   // WARNING[392] : warning392
   // WARNING[393] : warning393
   // WARNING[394] : warning394
   // WARNING[395] : warning395
   // WARNING[396] : warning396
   // WARNING[397] : warning397
   // WARNING[398] : warning398
   // WARNING[399] : warning399
   // WARNING[400] : warning400
   // WARNING[401] : warning401
   // WARNING[402] : warning402
   // WARNING[403] : warning403
   // WARNING[404] : warning404
   // WARNING[405] : warning405
   // WARNING[406] : warning406
   // WARNING[407] : warning407
   // WARNING[408] : warning408
   // WARNING[409] : warning409
   // WARNING[410] : warning410
   // WARNING[411] : warning411
   // WARNING[412] : warning412
   // WARNING[413] : warning413
   // WARNING[414] : warning414
   // WARNING[415] : warning415
   // WARNING[416] : warning416
   // WARNING[417] : Kistler +M01-KF121 Sensortest
   // WARNING[418] : Kistler +M01-KF121 Setup mismatch
   // WARNING[419] : Kistler +M01-KF121 NOK in Sequence
   // WARNING[420] : Kistler +M01-KF121 lost Cycles
   // WARNING[421] : Kistler +M01-KF121 Envelope
   // WARNING[422] : Kistler +M01-KF121 Samba no Network
   // WARNING[423] : Kistler +M01-KF121 Samba Memory Full
   // WARNING[424] : Kistler +M01-KF121 Memory Card Full
   // WARNING[425] : Kistler +M01-KF121 FIFO Full
   // WARNING[426] : Kistler +M01-KF121 Bereit fehlt
   // WARNING[427] : Kistler +M01-KF121 Bremsentest bei nächsten Füge-Start
   // WARNING[428] : Kistler +M01-KF121
   // WARNING[429] : warning429
   // WARNING[430] : warning430
   // WARNING[431] : warning431
   // WARNING[432] : warning432
   // WARNING[433] : Kistler +M01-KF122 Sensortest
   // WARNING[434] : Kistler +M01-KF122 Setup mismatch
   // WARNING[435] : Kistler +M01-KF122 NOK in Sequence
   // WARNING[436] : Kistler +M01-KF122 lost Cycles
   // WARNING[437] : Kistler +M01-KF122 Envelope
   // WARNING[438] : Kistler +M01-KF122 Samba no Network
   // WARNING[439] : Kistler +M01-KF122 Samba Memory Full
   // WARNING[440] : Kistler +M01-KF122 Memory Card Full
   // WARNING[441] : Kistler +M01-KF122 FIFO Full
   // WARNING[442] : Kistler +M01-KF122 Bereit fehlt
   // WARNING[443] : Kistler +M01-KF122 Bremsentest bei nächsten Füge-Start
   // WARNING[444] : Kistler +M01-KF122
   // WARNING[445] : warning445
   // WARNING[446] : warning446
   // WARNING[447] : warning447
   // WARNING[448] : warning448
   // WARNING[449] : Kistler +M01-KF123 Sensortest
   // WARNING[450] : Kistler +M01-KF123 Setup mismatch
   // WARNING[451] : Kistler +M01-KF123 NOK in Sequence
   // WARNING[452] : Kistler +M01-KF123 lost Cycles
   // WARNING[453] : Kistler +M01-KF123 Envelope
   // WARNING[454] : Kistler +M01-KF123 Samba no Network
   // WARNING[455] : Kistler +M01-KF123 Samba Memory Full
   // WARNING[456] : Kistler +M01-KF123 Memory Card Full
   // WARNING[457] : Kistler +M01-KF123 FIFO Full
   // WARNING[458] : Kistler +M01-KF123 Bereit fehlt
   // WARNING[459] : Kistler +M01-KF123 Bremsentest bei nächsten Füge-Start
   // WARNING[460] : Kistler +M01-KF123
   // WARNING[461] : warning461
   // WARNING[462] : warning462
   // WARNING[463] : warning463
   // WARNING[464] : warning464
   // WARNING[465] : Kistler +M01-KF124 Sensortest
   // WARNING[466] : Kistler +M01-KF124 Setup mismatch
   // WARNING[467] : Kistler +M01-KF124 NOK in Sequence
   // WARNING[468] : Kistler +M01-KF124 lost Cycles
   // WARNING[469] : Kistler +M01-KF124 Envelope
   // WARNING[470] : Kistler +M01-KF124 Samba no Network
   // WARNING[471] : Kistler +M01-KF124 Samba Memory Full
   // WARNING[472] : Kistler +M01-KF124 Memory Card Full
   // WARNING[473] : Kistler +M01-KF124 FIFO Full
   // WARNING[474] : Kistler +M01-KF124 Bereit fehlt
   // WARNING[475] : Kistler +M01-KF124 Bremsentest bei nächsten Füge-Start
   // WARNING[476] : Kistler +M01-KF124
   // WARNING[477] : warning477
   // WARNING[478] : warning478
   // WARNING[479] : warning479
   // WARNING[480] : warning480
   // WARNING[481] : Kistler +M01-KF125 Sensortest
   // WARNING[482] : Kistler +M01-KF125 Setup mismatch
   // WARNING[483] : Kistler +M01-KF125 NOK in Sequence
   // WARNING[484] : Kistler +M01-KF125 lost Cycles
   // WARNING[485] : Kistler +M01-KF125 Envelope
   // WARNING[486] : Kistler +M01-KF125 Samba no Network
   // WARNING[487] : Kistler +M01-KF125 Samba Memory Full
   // WARNING[488] : Kistler +M01-KF125 Memory Card Full
   // WARNING[489] : Kistler +M01-KF125 FIFO Full
   // WARNING[490] : Kistler +M01-KF125 Bereit fehlt
   // WARNING[491] : Kistler +M01-KF125 Bremsentest bei nächsten Füge-Start
   // WARNING[492] : Kistler +M01-KF125
   // WARNING[493] : warning493
   // WARNING[494] : warning494
   // WARNING[495] : warning495
   // WARNING[496] : warning496
   // WARNING[497] : Kistler +M01-KF126 Sensortest
   // WARNING[498] : Kistler +M01-KF126 Setup mismatch
   // WARNING[499] : Kistler +M01-KF126 NOK in Sequence
   // WARNING[500] : Kistler +M01-KF126 lost Cycles
   // WARNING[501] : Kistler +M01-KF126 Envelope
   // WARNING[502] : Kistler +M01-KF126 Samba no Network
   // WARNING[503] : Kistler +M01-KF126 Samba Memory Full
   // WARNING[504] : Kistler +M01-KF126 Memory Card Full
   // WARNING[505] : Kistler +M01-KF126 FIFO Full
   // WARNING[506] : Kistler +M01-KF126 Bereit fehlt
   // WARNING[507] : Kistler +M01-KF126 Bremsentest bei nächsten Füge-Start
   // WARNING[508] : Kistler +M01-KF126
   // WARNING[509] : warning509
   // WARNING[510] : warning510
   // WARNING[511] : warning511
   // WARNING[512] : warning512
END_DATA_BLOCK
